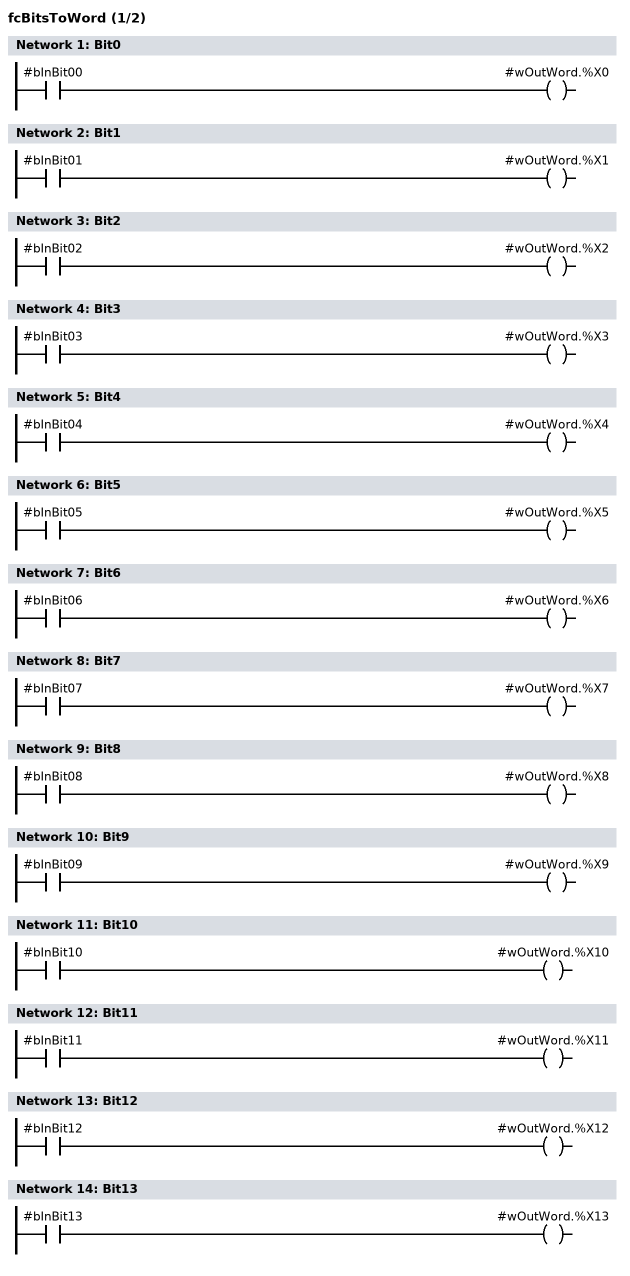
   RUNG wire#powerrail
      Contact( #bInBit00 )
      Coil( #wOutWord.%X0 )
   END_RUNG
   // the same network as SCL:
   #wOutWord.%X0 := #bInBit00;
END_REGION

REGION Network 2: Bit1
   RUNG wire#powerrail
      Contact( #bInBit01 )
      Coil( #wOutWord.%X1 )
   END_RUNG
   // the same network as SCL:
   #wOutWord.%X1 := #bInBit01;
END_REGION

REGION Network 3: Bit2
   RUNG wire#powerrail
      Contact( #bInBit02 )
      Coil( #wOutWord.%X2 )
   END_RUNG
   // the same network as SCL:
   #wOutWord.%X2 := #bInBit02;
END_REGION

REGION Network 4: Bit3
   RUNG wire#powerrail
      Contact( #bInBit03 )
      Coil( #wOutWord.%X3 )
   END_RUNG
   // the same network as SCL:
   #wOutWord.%X3 := #bInBit03;
END_REGION

REGION Network 5: Bit4
   RUNG wire#powerrail
      Contact( #bInBit04 )
      Coil( #wOutWord.%X4 )
   END_RUNG
   // the same network as SCL:
   #wOutWord.%X4 := #bInBit04;
END_REGION

REGION Network 6: Bit5
   RUNG wire#powerrail
      Contact( #bInBit05 )
      Coil( #wOutWord.%X5 )
   END_RUNG
   // the same network as SCL:
   #wOutWord.%X5 := #bInBit05;
END_REGION

REGION Network 7: Bit6
   RUNG wire#powerrail
      Contact( #bInBit06 )
      Coil( #wOutWord.%X6 )
   END_RUNG
   // the same network as SCL:
   #wOutWord.%X6 := #bInBit06;
END_REGION

REGION Network 8: Bit7
   RUNG wire#powerrail
      Contact( #bInBit07 )
      Coil( #wOutWord.%X7 )
   END_RUNG
   // the same network as SCL:
   #wOutWord.%X7 := #bInBit07;
END_REGION

REGION Network 9: Bit8
   RUNG wire#powerrail
      Contact( #bInBit08 )
      Coil( #wOutWord.%X8 )
   END_RUNG
   // the same network as SCL:
   #wOutWord.%X8 := #bInBit08;
END_REGION

REGION Network 10: Bit9
   RUNG wire#powerrail
      Contact( #bInBit09 )
      Coil( #wOutWord.%X9 )
   END_RUNG
   // the same network as SCL:
   #wOutWord.%X9 := #bInBit09;
END_REGION

REGION Network 11: Bit10
   RUNG wire#powerrail
      Contact( #bInBit10 )
      Coil( #wOutWord.%X10 )
   END_RUNG
   // the same network as SCL:
   #wOutWord.%X10 := #bInBit10;
END_REGION

REGION Network 12: Bit11
   RUNG wire#powerrail
      Contact( #bInBit11 )
      Coil( #wOutWord.%X11 )
   END_RUNG
   // the same network as SCL:
   #wOutWord.%X11 := #bInBit11;
END_REGION

REGION Network 13: Bit12
   RUNG wire#powerrail
      Contact( #bInBit12 )
      Coil( #wOutWord.%X12 )
   END_RUNG
   // the same network as SCL:
   #wOutWord.%X12 := #bInBit12;
END_REGION

REGION Network 14: Bit13
   RUNG wire#powerrail
      Contact( #bInBit13 )
      Coil( #wOutWord.%X13 )
   END_RUNG
   // the same network as SCL:
   #wOutWord.%X13 := #bInBit13;
END_REGION

REGION Network 15: Bit14
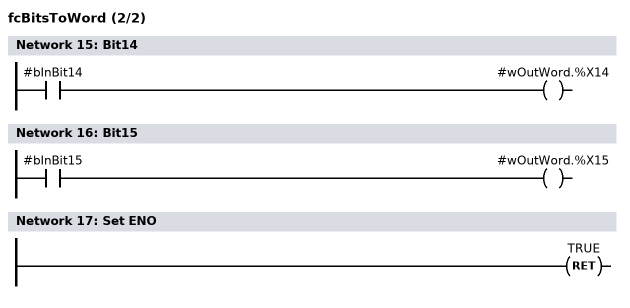
   RUNG wire#powerrail
      Contact( #bInBit14 )
      Coil( #wOutWord.%X14 )
   END_RUNG
   // the same network as SCL:
   #wOutWord.%X14 := #bInBit14;
END_REGION

REGION Network 16: Bit15
   RUNG wire#powerrail
      Contact( #bInBit15 )
      Coil( #wOutWord.%X15 )
   END_RUNG
   // the same network as SCL:
   #wOutWord.%X15 := #bInBit15;
END_REGION

REGION Network 17: Set ENO
   RUNG wire#powerrail
      ReturnCoil( TRUE )
   END_RUNG
   // the same network as SCL:
   ENO := TRUE;
   RETURN;
END_REGION
END_FUNCTION

FUNCTION "fcWordToBits" : Void   // FC303, LAD
TITLE = Breaks A Word Into Individual Bits
{ S7_Optimized_Access := 'TRUE' }
AUTHOR : DMC
FAMILY : LowLevel
VERSION : 0.1
   VAR_INPUT
      wInWord : Word;   // Word to be broken into individual bits
   END_VAR
   VAR_OUTPUT
      bOutBit00 : Bool;   // Bit 0
      bOutBit01 : Bool;   // Bit 1
      bOutBit02 : Bool;   // Bit 2
      bOutBit03 : Bool;   // Bit 3
      bOutBit04 : Bool;   // Bit 4
      bOutBit05 : Bool;   // Bit 5
      bOutBit06 : Bool;   // Bit 6
      bOutBit07 : Bool;   // Bit 7
      bOutBit08 : Bool;   // Bit 8
      bOutBit09 : Bool;   // Bit 9
      bOutBit10 : Bool;   // Bit 10
      bOutBit11 : Bool;   // Bit 11
      bOutBit12 : Bool;   // Bit 12
      bOutBit13 : Bool;   // Bit 13
      bOutBit14 : Bool;   // Bit 14
      bOutBit15 : Bool;   // Bit 15
   END_VAR
BEGIN

REGION Network 1: Bit0
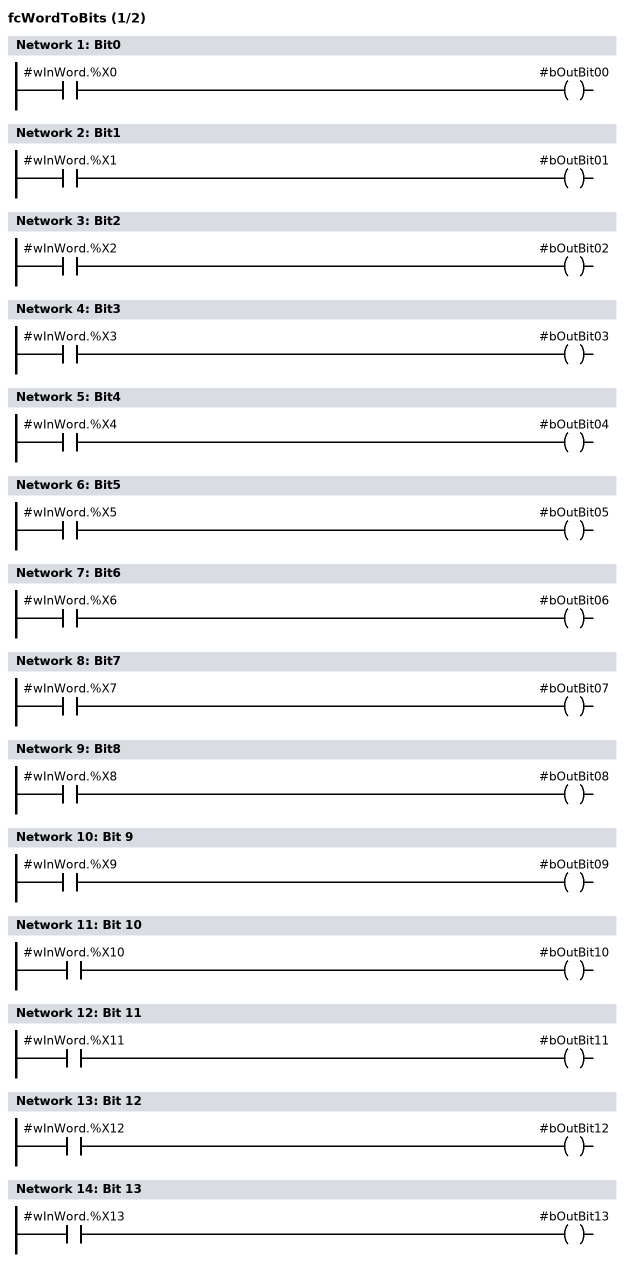
   RUNG wire#powerrail
      Contact( #wInWord.%X0 )
      Coil( #bOutBit00 )
   END_RUNG
   // the same network as SCL:
   #bOutBit00 := #wInWord.%X0;
END_REGION

REGION Network 2: Bit1
   RUNG wire#powerrail
      Contact( #wInWord.%X1 )
      Coil( #bOutBit01 )
   END_RUNG
   // the same network as SCL:
   #bOutBit01 := #wInWord.%X1;
END_REGION

REGION Network 3: Bit2
   RUNG wire#powerrail
      Contact( #wInWord.%X2 )
      Coil( #bOutBit02 )
   END_RUNG
   // the same network as SCL:
   #bOutBit02 := #wInWord.%X2;
END_REGION

REGION Network 4: Bit3
   RUNG wire#powerrail
      Contact( #wInWord.%X3 )
      Coil( #bOutBit03 )
   END_RUNG
   // the same network as SCL:
   #bOutBit03 := #wInWord.%X3;
END_REGION

REGION Network 5: Bit4
   RUNG wire#powerrail
      Contact( #wInWord.%X4 )
      Coil( #bOutBit04 )
   END_RUNG
   // the same network as SCL:
   #bOutBit04 := #wInWord.%X4;
END_REGION

REGION Network 6: Bit5
   RUNG wire#powerrail
      Contact( #wInWord.%X5 )
      Coil( #bOutBit05 )
   END_RUNG
   // the same network as SCL:
   #bOutBit05 := #wInWord.%X5;
END_REGION

REGION Network 7: Bit6
   RUNG wire#powerrail
      Contact( #wInWord.%X6 )
      Coil( #bOutBit06 )
   END_RUNG
   // the same network as SCL:
   #bOutBit06 := #wInWord.%X6;
END_REGION

REGION Network 8: Bit7
   RUNG wire#powerrail
      Contact( #wInWord.%X7 )
      Coil( #bOutBit07 )
   END_RUNG
   // the same network as SCL:
   #bOutBit07 := #wInWord.%X7;
END_REGION

REGION Network 9: Bit8
   RUNG wire#powerrail
      Contact( #wInWord.%X8 )
      Coil( #bOutBit08 )
   END_RUNG
   // the same network as SCL:
   #bOutBit08 := #wInWord.%X8;
END_REGION

REGION Network 10: Bit 9
   RUNG wire#powerrail
      Contact( #wInWord.%X9 )
      Coil( #bOutBit09 )
   END_RUNG
   // the same network as SCL:
   #bOutBit09 := #wInWord.%X9;
END_REGION

REGION Network 11: Bit 10
   RUNG wire#powerrail
      Contact( #wInWord.%X10 )
      Coil( #bOutBit10 )
   END_RUNG
   // the same network as SCL:
   #bOutBit10 := #wInWord.%X10;
END_REGION

REGION Network 12: Bit 11
   RUNG wire#powerrail
      Contact( #wInWord.%X11 )
      Coil( #bOutBit11 )
   END_RUNG
   // the same network as SCL:
   #bOutBit11 := #wInWord.%X11;
END_REGION

REGION Network 13: Bit 12
   RUNG wire#powerrail
      Contact( #wInWord.%X12 )
      Coil( #bOutBit12 )
   END_RUNG
   // the same network as SCL:
   #bOutBit12 := #wInWord.%X12;
END_REGION

REGION Network 14: Bit 13
   RUNG wire#powerrail
      Contact( #wInWord.%X13 )
      Coil( #bOutBit13 )
   END_RUNG
   // the same network as SCL:
   #bOutBit13 := #wInWord.%X13;
END_REGION

REGION Network 15: Bit 14
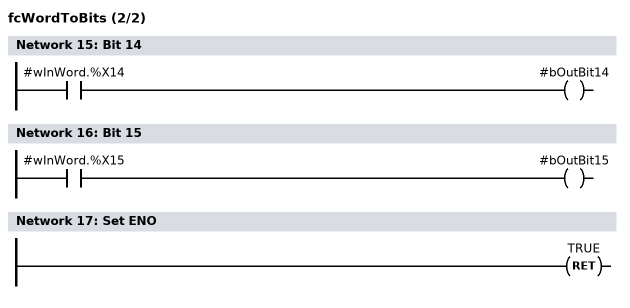
   RUNG wire#powerrail
      Contact( #wInWord.%X14 )
      Coil( #bOutBit14 )
   END_RUNG
   // the same network as SCL:
   #bOutBit14 := #wInWord.%X14;
END_REGION

REGION Network 16: Bit 15
   RUNG wire#powerrail
      Contact( #wInWord.%X15 )
      Coil( #bOutBit15 )
   END_RUNG
   // the same network as SCL:
   #bOutBit15 := #wInWord.%X15;
END_REGION

REGION Network 17: Set ENO
   RUNG wire#powerrail
      ReturnCoil( TRUE )
   END_RUNG
   // the same network as SCL:
   ENO := TRUE;
   RETURN;
END_REGION
END_FUNCTION

// folder: Resources/fbVFD/Resources/HMI

FUNCTION_BLOCK "fbErrorScroller"   // FB330, LAD
TITLE = Scrolls through the error codes for display on the HMI
{ S7_Optimized_Access := 'TRUE' }
AUTHOR : DMC
FAMILY : Error
VERSION : 0.1
   VAR_INPUT
      bInError01 : Bool;   // Error 1 In Error Array
      bInError02 : Bool;   // Error 2 In Error Array
      bInError03 : Bool;   // Error 3 In Error Array
      bInError04 : Bool;   // Error 4 In Error Array
      bInError05 : Bool;   // Error 5 In Error Array
      bInError06 : Bool;   // Error 6 In Error Array
      bInError07 : Bool;   // Error 7 In Error Array
      bInError08 : Bool;   // Error 8 In Error Array
      bInError09 : Bool;   // Error 9 In Error Array
      bInError10 : Bool;   // Error 10 In Error Array
      bInError11 : Bool;   // Error 11 In Error Array
      bInError12 : Bool;   // Error 12 In Error Array
      bInError13 : Bool;   // Error 13 In Error Array
      bInError14 : Bool;   // Error 14 In Error Array
      bInError15 : Bool;   // Error 15 In Error Array
      bInError16 : Bool;   // Error 16 In Error Array
      bInError17 : Bool;   // Error 17 In Error Array
      bInError18 : Bool;   // Error 18 In Error Array
      bInError19 : Bool;   // Error 19 In Error Array
      bInError20 : Bool;   // Error 20 In Error Array
      bInError21 : Bool;   // Error 21 In Error Array
      bInError22 : Bool;   // Error 22 In Error Array
      bInError23 : Bool;   // Error 23 In Error Array
      bInError24 : Bool;   // Error 24 In Error Array
      bInError25 : Bool;   // Error 25 In Error Array
      bInError26 : Bool;   // Error 26 In Error Array
      bInError27 : Bool;   // Error 27 In Error Array
      bInError28 : Bool;   // Error 28 In Error Array
      bInError29 : Bool;   // Error 29 In Error Array
      bInError30 : Bool;   // Error 30 In Error Array
   END_VAR
   VAR_OUTPUT
      bOutErrorExists : Bool;   // An Error Exists
      iOutScrollingErrorNumber : Int;   // Current Index when scrolling through errors
   END_VAR
   VAR
      TON_ErrorDelay : TON_TIME;   // Delay between each scroll for a new error
      abErrors : Array[#ciIndexLow..#ciIndexHigh] of Bool;
      iNextScrollNum : Int := 1;   // Index of next error position
      iErrorsScrollNum : Int := 1;   // Index of current error position
      bScrolling : Bool;   // Indicates we are scrolling
      bTON_ErrorDelay : Bool;
   END_VAR
   VAR_TEMP
      bErrorExists : Bool;   // Error Exists
   END_VAR
   VAR CONSTANT
      ciNoErrrors : Int := 0;
      ciIndexLow : Int := 1;
      ciIndexHigh : Int := 30;
   END_VAR
   VAR_TEMP   // added for the SCL form of the ladder/FBD networks
      _w1 : Bool;
   END_VAR
BEGIN

REGION Network 1: Check for valid array indexes
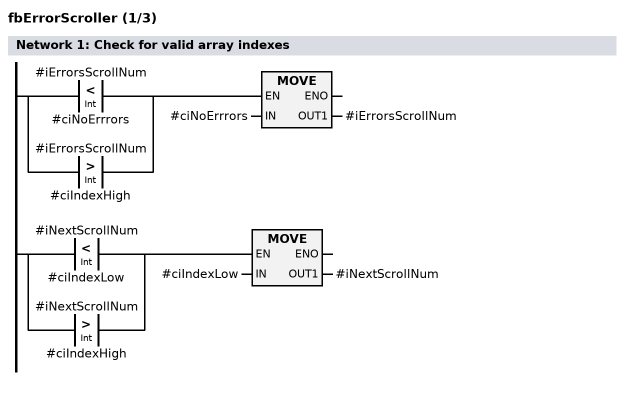
   RUNG wire#powerrail
      { S7_Templates := "SrcType := Int" } LT_Contact(in1 := #iErrorsScrollNum, in2 := #ciNoErrrors)
      wire#w1
      Move(in := #ciNoErrrors, out1 => #iErrorsScrollNum)
   END_RUNG
   RUNG wire#powerrail
      { S7_Templates := "SrcType := Int" } GT_Contact(in1 := #iErrorsScrollNum, in2 := #ciIndexHigh)
   END_RUNG wire#w1
   RUNG wire#powerrail
      { S7_Templates := "SrcType := Int" } LT_Contact(in1 := #iNextScrollNum, in2 := #ciIndexLow)
      wire#w2
      Move(in := #ciIndexLow, out1 => #iNextScrollNum)
   END_RUNG
   RUNG wire#powerrail
      { S7_Templates := "SrcType := Int" } GT_Contact(in1 := #iNextScrollNum, in2 := #ciIndexHigh)
   END_RUNG wire#w2
   // the same network as SCL:
   IF (#iErrorsScrollNum < #ciNoErrrors) OR (#iErrorsScrollNum > #ciIndexHigh) THEN
       #iErrorsScrollNum := #ciNoErrrors;
   END_IF;
   IF (#iNextScrollNum < #ciIndexLow) OR (#iNextScrollNum > #ciIndexHigh) THEN
       #iNextScrollNum := #ciIndexLow;
   END_IF;
END_REGION

REGION Network 2: Check if error exists
   // OR all of the possible errors. If any error Exists, SET bErrorExists
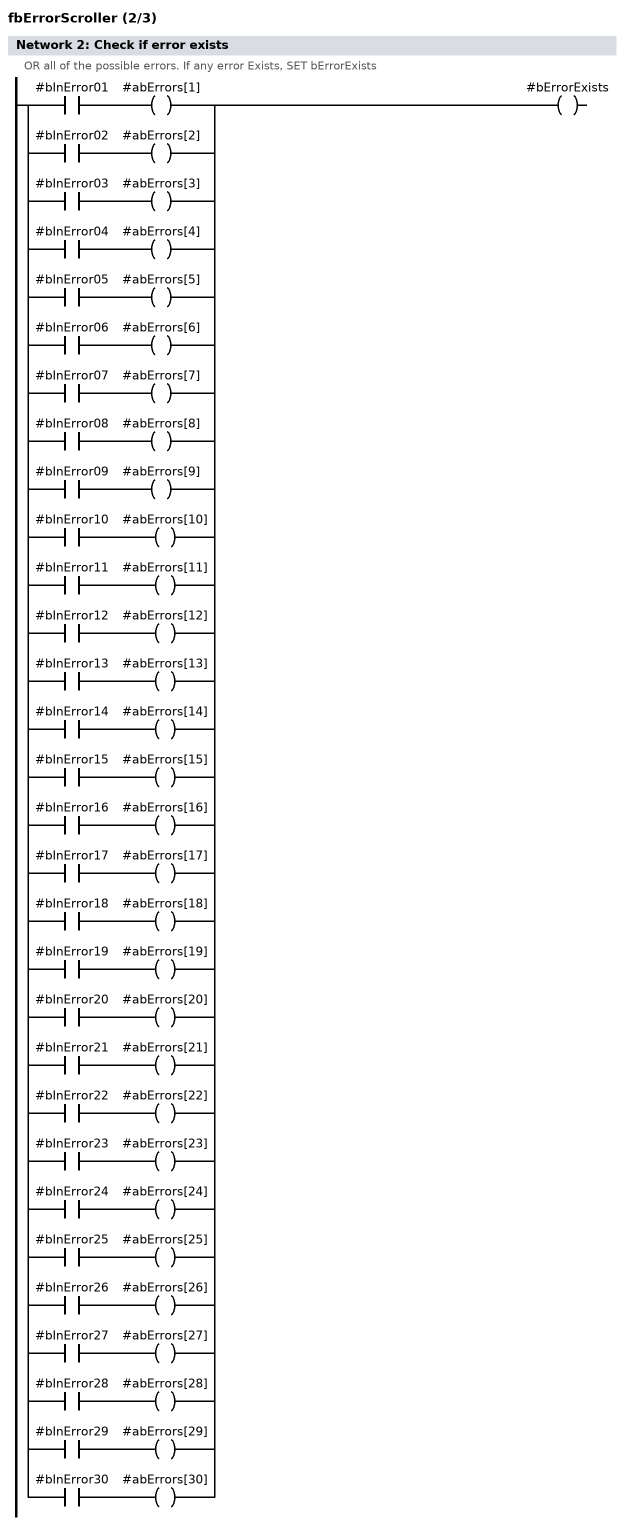
   RUNG wire#powerrail
      Contact( #bInError01 )
      Coil( #abErrors[1] )
      wire#w1
      Coil( #bErrorExists )
   END_RUNG
   RUNG wire#powerrail
      Contact( #bInError02 )
      Coil( #abErrors[2] )
   END_RUNG wire#w1
   RUNG wire#powerrail
      Contact( #bInError03 )
      Coil( #abErrors[3] )
   END_RUNG wire#w1
   RUNG wire#powerrail
      Contact( #bInError04 )
      Coil( #abErrors[4] )
   END_RUNG wire#w1
   RUNG wire#powerrail
      Contact( #bInError05 )
      Coil( #abErrors[5] )
   END_RUNG wire#w1
   RUNG wire#powerrail
      Contact( #bInError06 )
      Coil( #abErrors[6] )
   END_RUNG wire#w1
   RUNG wire#powerrail
      Contact( #bInError07 )
      Coil( #abErrors[7] )
   END_RUNG wire#w1
   RUNG wire#powerrail
      Contact( #bInError08 )
      Coil( #abErrors[8] )
   END_RUNG wire#w1
   RUNG wire#powerrail
      Contact( #bInError09 )
      Coil( #abErrors[9] )
   END_RUNG wire#w1
   RUNG wire#powerrail
      Contact( #bInError10 )
      Coil( #abErrors[10] )
   END_RUNG wire#w1
   RUNG wire#powerrail
      Contact( #bInError11 )
      Coil( #abErrors[11] )
   END_RUNG wire#w1
   RUNG wire#powerrail
      Contact( #bInError12 )
      Coil( #abErrors[12] )
   END_RUNG wire#w1
   RUNG wire#powerrail
      Contact( #bInError13 )
      Coil( #abErrors[13] )
   END_RUNG wire#w1
   RUNG wire#powerrail
      Contact( #bInError14 )
      Coil( #abErrors[14] )
   END_RUNG wire#w1
   RUNG wire#powerrail
      Contact( #bInError15 )
      Coil( #abErrors[15] )
   END_RUNG wire#w1
   RUNG wire#powerrail
      Contact( #bInError16 )
      Coil( #abErrors[16] )
   END_RUNG wire#w1
   RUNG wire#powerrail
      Contact( #bInError17 )
      Coil( #abErrors[17] )
   END_RUNG wire#w1
   RUNG wire#powerrail
      Contact( #bInError18 )
      Coil( #abErrors[18] )
   END_RUNG wire#w1
   RUNG wire#powerrail
      Contact( #bInError19 )
      Coil( #abErrors[19] )
   END_RUNG wire#w1
   RUNG wire#powerrail
      Contact( #bInError20 )
      Coil( #abErrors[20] )
   END_RUNG wire#w1
   RUNG wire#powerrail
      Contact( #bInError21 )
      Coil( #abErrors[21] )
   END_RUNG wire#w1
   RUNG wire#powerrail
      Contact( #bInError22 )
      Coil( #abErrors[22] )
   END_RUNG wire#w1
   RUNG wire#powerrail
      Contact( #bInError23 )
      Coil( #abErrors[23] )
   END_RUNG wire#w1
   RUNG wire#powerrail
      Contact( #bInError24 )
      Coil( #abErrors[24] )
   END_RUNG wire#w1
   RUNG wire#powerrail
      Contact( #bInError25 )
      Coil( #abErrors[25] )
   END_RUNG wire#w1
   RUNG wire#powerrail
      Contact( #bInError26 )
      Coil( #abErrors[26] )
   END_RUNG wire#w1
   RUNG wire#powerrail
      Contact( #bInError27 )
      Coil( #abErrors[27] )
   END_RUNG wire#w1
   RUNG wire#powerrail
      Contact( #bInError28 )
      Coil( #abErrors[28] )
   END_RUNG wire#w1
   RUNG wire#powerrail
      Contact( #bInError29 )
      Coil( #abErrors[29] )
   END_RUNG wire#w1
   RUNG wire#powerrail
      Contact( #bInError30 )
      Coil( #abErrors[30] )
   END_RUNG wire#w1
   // the same network as SCL:
   #abErrors[1] := #bInError01;
   #abErrors[2] := #bInError02;
   #abErrors[3] := #bInError03;
   #abErrors[4] := #bInError04;
   #abErrors[5] := #bInError05;
   #abErrors[6] := #bInError06;
   #abErrors[7] := #bInError07;
   #abErrors[8] := #bInError08;
   #abErrors[9] := #bInError09;
   #abErrors[10] := #bInError10;
   #abErrors[11] := #bInError11;
   #abErrors[12] := #bInError12;
   #abErrors[13] := #bInError13;
   #abErrors[14] := #bInError14;
   #abErrors[15] := #bInError15;
   #abErrors[16] := #bInError16;
   #abErrors[17] := #bInError17;
   #abErrors[18] := #bInError18;
   #abErrors[19] := #bInError19;
   #abErrors[20] := #bInError20;
   #abErrors[21] := #bInError21;
   #abErrors[22] := #bInError22;
   #abErrors[23] := #bInError23;
   #abErrors[24] := #bInError24;
   #abErrors[25] := #bInError25;
   #abErrors[26] := #bInError26;
   #abErrors[27] := #bInError27;
   #abErrors[28] := #bInError28;
   #abErrors[29] := #bInError29;
   #abErrors[30] := #bInError30;
   #bErrorExists := #bInError01 OR #bInError02 OR #bInError03 OR #bInError04 OR #bInError05 OR #bInError06 OR #bInError07 OR #bInError08 OR #bInError09 OR #bInError10 OR #bInError11 OR #bInError12 OR #bInError13 OR #bInError14 OR #bInError15 OR #bInError16 OR #bInError17 OR #bInError18 OR #bInError19 OR #bInError20 OR #bInError21 OR #bInError22 OR #bInError23 OR #bInError24 OR #bInError25 OR #bInError26 OR #bInError27 OR #bInError28 OR #bInError29 OR #bInError30;
END_REGION

REGION Network 3: Timer to change displayed error
   // ============================ Scroll errors on HMI ========================
   // Timed delay
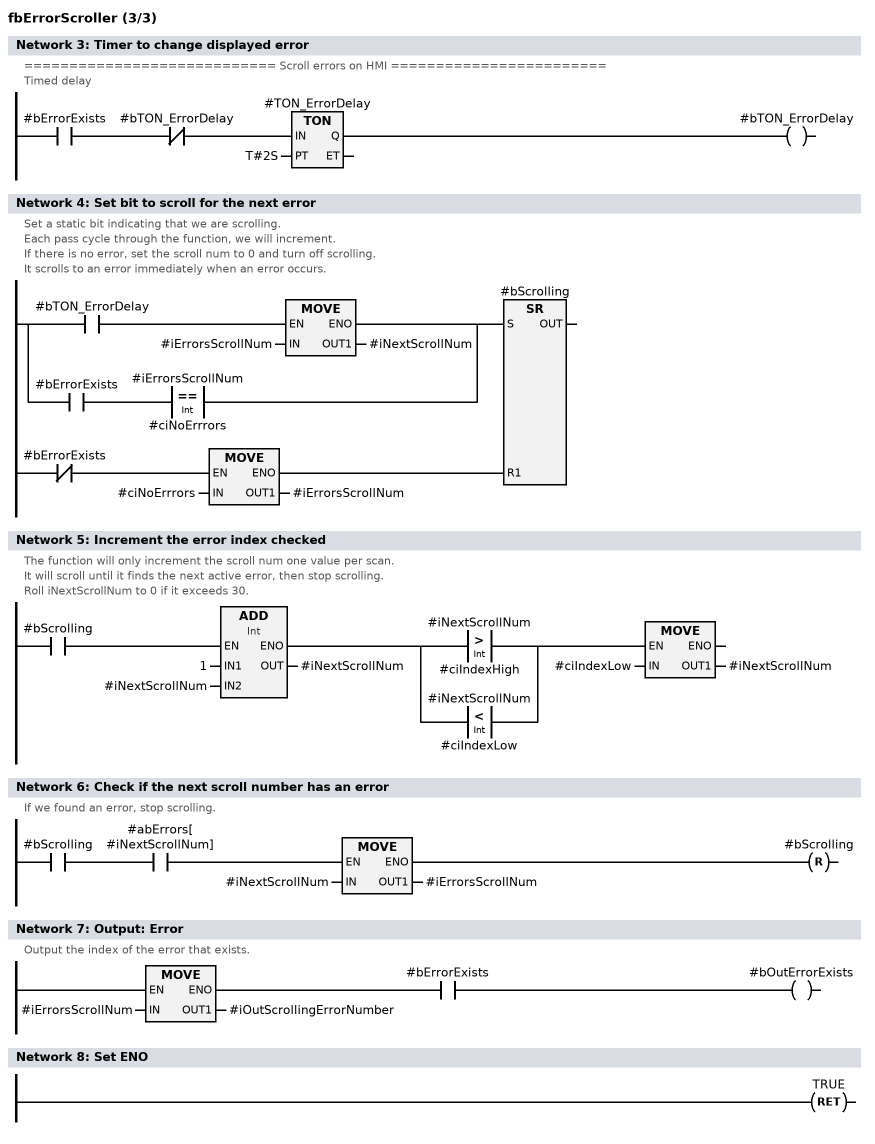
   #TON_ErrorDelay(IN := #bErrorExists AND NOT #bTON_ErrorDelay, PT := T#2S);   // TON
   #bTON_ErrorDelay := #TON_ErrorDelay.Q;
END_REGION

REGION Network 4: Set bit to scroll for the next error
   // Set a static bit indicating that we are scrolling.  
   // Each pass cycle through the function, we will increment.  
   // If there is no error, set the scroll num to 0 and turn off scrolling.  
   // It scrolls to an error immediately when an error occurs.
   RUNG wire#powerrail
      Contact( #bTON_ErrorDelay )
      { S7_GenerateENO := "TRUE" } Move(in := #iErrorsScrollNum, out1 => #iNextScrollNum)
      wire#w1
      S_SR(operand := #bScrolling, r1 := wire#w2)
   END_RUNG
   RUNG wire#powerrail
      Contact( #bErrorExists )
      { S7_Templates := "SrcType := Int" } EQ_Contact(in1 := #iErrorsScrollNum, in2 := #ciNoErrrors)
   END_RUNG wire#w1
   RUNG wire#powerrail
      I_Contact( #bErrorExists )
      { S7_GenerateENO := "TRUE" } Move(in := #ciNoErrrors, out1 => #iErrorsScrollNum)
   END_RUNG wire#w2
   // the same network as SCL:
   // ENO of a box is taken as its EN; it also drops when the box reports an error
   IF #bTON_ErrorDelay THEN #iNextScrollNum := #iErrorsScrollNum; END_IF;
   #_w1 := #bTON_ErrorDelay OR (#bErrorExists AND (#iErrorsScrollNum = #ciNoErrrors));
   IF NOT #bErrorExists THEN #iErrorsScrollNum := #ciNoErrrors; END_IF;
   IF #_w1 THEN
       #bScrolling := TRUE;   // SR flip-flop
   END_IF;
   IF NOT #bErrorExists THEN #bScrolling := FALSE; END_IF;
END_REGION

REGION Network 5: Increment the error index checked
   // The function will only increment the scroll num one value per scan.  
   // It will scroll until it finds the next active error, then stop scrolling.  
   // Roll iNextScrollNum to 0 if it exceeds 30.
   RUNG wire#powerrail
      Contact( #bScrolling )
      { S7_Templates := "SrcType := Int"; S7_GenerateENO := "TRUE" } Add(in1 := 1, in2 := #iNextScrollNum, out => #iNextScrollNum)
      wire#w1
      { S7_Templates := "SrcType := Int" } GT_Contact(in1 := #iNextScrollNum, in2 := #ciIndexHigh)
      wire#w2
      { S7_GenerateENO := "TRUE" } Move(in := #ciIndexLow, out1 => #iNextScrollNum)
   END_RUNG
   RUNG wire#w1
      { S7_Templates := "SrcType := Int" } LT_Contact(in1 := #iNextScrollNum, in2 := #ciIndexLow)
   END_RUNG wire#w2
   // the same network as SCL:
   // ENO of a box is taken as its EN; it also drops when the box reports an error
   IF #bScrolling THEN #iNextScrollNum := 1 + #iNextScrollNum; END_IF;
   IF #bScrolling AND ((#iNextScrollNum > #ciIndexHigh) OR (#iNextScrollNum < #ciIndexLow)) THEN
       #iNextScrollNum := #ciIndexLow;
   END_IF;
END_REGION

REGION Network 6: Check if the next scroll number has an error
   // If we found an error, stop scrolling.
   RUNG wire#powerrail
      Contact( #bScrolling )
      Contact( #abErrors[#iNextScrollNum] )
      { S7_GenerateENO := "TRUE" } Move(in := #iNextScrollNum, out1 => #iErrorsScrollNum)
      R_Coil( #bScrolling )
   END_RUNG
   // the same network as SCL:
   // ENO of a box is taken as its EN; it also drops when the box reports an error
   IF #bScrolling AND #abErrors[#iNextScrollNum] THEN
       #iErrorsScrollNum := #iNextScrollNum;
       #bScrolling := FALSE;
   END_IF;
END_REGION

REGION Network 7: Output: Error
   // Output the index of the error that exists.
   RUNG wire#powerrail
      { S7_GenerateENO := "TRUE" } Move(in := #iErrorsScrollNum, out1 => #iOutScrollingErrorNumber)
      Contact( #bErrorExists )
      Coil( #bOutErrorExists )
   END_RUNG
   // the same network as SCL:
   // ENO of a box is taken as its EN; it also drops when the box reports an error
   #iOutScrollingErrorNumber := #iErrorsScrollNum;
   #bOutErrorExists := #bErrorExists;
END_REGION

REGION Network 8: Set ENO
   RUNG wire#powerrail
      ReturnCoil( TRUE )
   END_RUNG
   // the same network as SCL:
   ENO := TRUE;
   RETURN;
END_REGION
END_FUNCTION_BLOCK

FUNCTION "fcHMIBitEnable" : Void   // FC329, LAD
TITLE = Handles an async reading of an HMI bit to avoid race conditions, includes an enable bit
{ S7_Optimized_Access := 'TRUE' }
VERSION : 0.1
   VAR_INPUT
      bInToggle : Bool;
      bInLatch : Bool;
      bInEnable : Bool;
   END_VAR
   VAR_OUTPUT
      bOutEnable : Bool;
   END_VAR
   VAR_IN_OUT
      bInOutHMI : Bool;
      bInOutPLC : Bool;
   END_VAR
   VAR_TEMP   // added for the SCL form of the ladder/FBD networks
      _w1 : Bool;
   END_VAR
BEGIN

REGION Network 1: If not latching or toggling, reset the PLC bit every scan
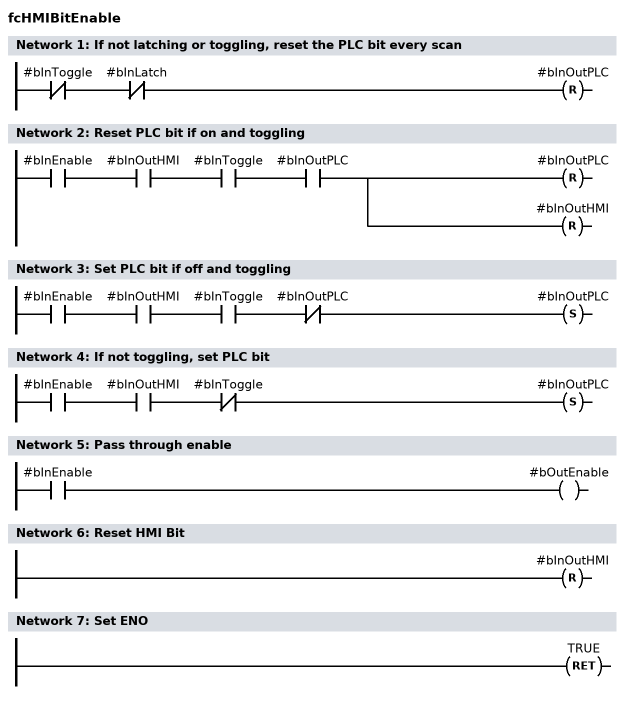
   RUNG wire#powerrail
      I_Contact( #bInToggle )
      I_Contact( #bInLatch )
      R_Coil( #bInOutPLC )
   END_RUNG
   // the same network as SCL:
   IF NOT #bInToggle AND NOT #bInLatch THEN #bInOutPLC := FALSE; END_IF;
END_REGION

REGION Network 2: Reset PLC bit if on and toggling
   RUNG wire#powerrail
      Contact( #bInEnable )
      Contact( #bInOutHMI )
      Contact( #bInToggle )
      Contact( #bInOutPLC )
      wire#w1
      R_Coil( #bInOutPLC )
   END_RUNG
   RUNG wire#w1
      R_Coil( #bInOutHMI )
   END_RUNG
   // the same network as SCL:
   #_w1 := #bInEnable AND #bInOutHMI AND #bInToggle AND #bInOutPLC;
   IF #_w1 THEN
       #bInOutPLC := FALSE;
       #bInOutHMI := FALSE;
   END_IF;
END_REGION

REGION Network 3: Set PLC bit if off and toggling
   RUNG wire#powerrail
      Contact( #bInEnable )
      Contact( #bInOutHMI )
      Contact( #bInToggle )
      I_Contact( #bInOutPLC )
      S_Coil( #bInOutPLC )
   END_RUNG
   // the same network as SCL:
   IF #bInEnable AND #bInOutHMI AND #bInToggle AND NOT #bInOutPLC THEN #bInOutPLC := TRUE; END_IF;
END_REGION

REGION Network 4: If not toggling, set PLC bit
   RUNG wire#powerrail
      Contact( #bInEnable )
      Contact( #bInOutHMI )
      I_Contact( #bInToggle )
      S_Coil( #bInOutPLC )
   END_RUNG
   // the same network as SCL:
   IF #bInEnable AND #bInOutHMI AND NOT #bInToggle THEN #bInOutPLC := TRUE; END_IF;
END_REGION

REGION Network 5: Pass through enable
   RUNG wire#powerrail
      Contact( #bInEnable )
      Coil( #bOutEnable )
   END_RUNG
   // the same network as SCL:
   #bOutEnable := #bInEnable;
END_REGION

REGION Network 6: Reset HMI Bit
   RUNG wire#powerrail
      R_Coil( #bInOutHMI )
   END_RUNG
   // the same network as SCL:
   #bInOutHMI := FALSE;
END_REGION

REGION Network 7: Set ENO
   RUNG wire#powerrail
      ReturnCoil( TRUE )
   END_RUNG
   // the same network as SCL:
   ENO := TRUE;
   RETURN;
END_REGION
END_FUNCTION

FUNCTION "fcSetHMIStatusSimulation" : Void   // FC333, LAD
TITLE = Sets HMI Status
{ S7_Optimized_Access := 'TRUE' }
VERSION : 0.1
// Wrapper function for setting the HMI status of a device
// 
// In order of priority:
// 1. E-stop
// 2. Error
// 3. Forward/Work Position
// 4. Reverse/Home Position
// 5. Forward/Work On
// 6. Reverse/Home On
// 7. None
   VAR_INPUT
      bInEstop : Bool;
      bInError : Bool;
      bInForwardWork : Bool;
      bInReverseHome : Bool;
      bInOnForwardWork : Bool;
      bInOnReverseHome : Bool;
      bInSimulate : Bool;
   END_VAR
   VAR_OUTPUT
      iOutStatus : Int;
   END_VAR
BEGIN

REGION Network 1: Set Reverse/Home On
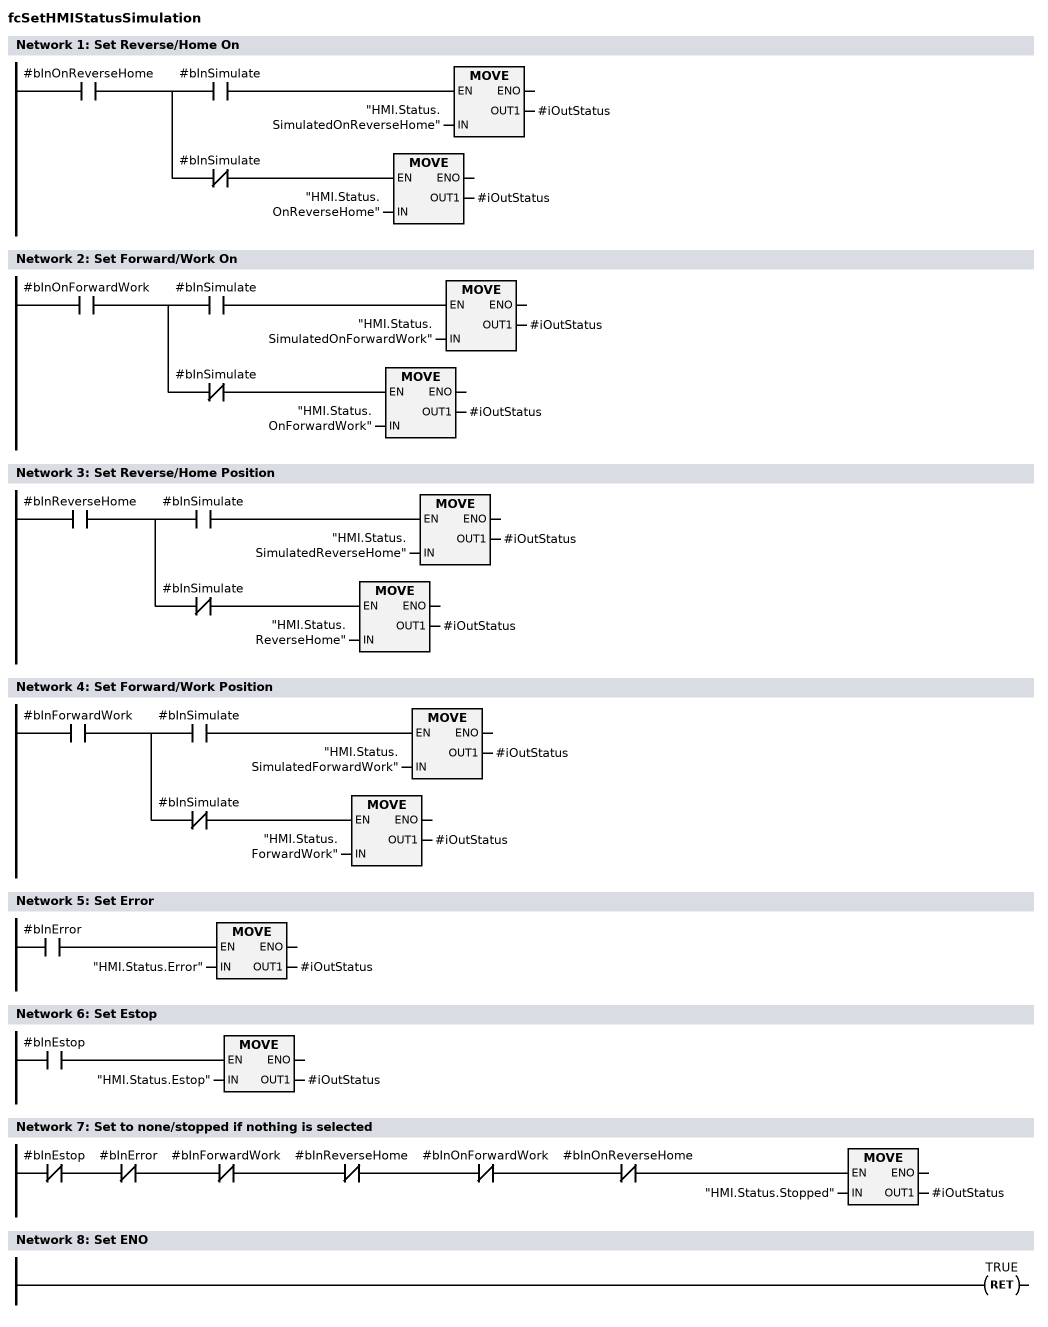
   RUNG wire#powerrail
      Contact( #bInOnReverseHome )
      wire#w1
      Contact( #bInSimulate )
      Move(in := "HMI.Status.SimulatedOnReverseHome", out1 => #iOutStatus)
   END_RUNG
   RUNG wire#w1
      I_Contact( #bInSimulate )
      Move(in := "HMI.Status.OnReverseHome", out1 => #iOutStatus)
   END_RUNG
   // the same network as SCL:
   IF #bInOnReverseHome AND #bInSimulate THEN #iOutStatus := "HMI.Status.SimulatedOnReverseHome"; END_IF;
   IF #bInOnReverseHome AND NOT #bInSimulate THEN #iOutStatus := "HMI.Status.OnReverseHome"; END_IF;
END_REGION

REGION Network 2: Set Forward/Work On
   RUNG wire#powerrail
      Contact( #bInOnForwardWork )
      wire#w1
      Contact( #bInSimulate )
      Move(in := "HMI.Status.SimulatedOnForwardWork", out1 => #iOutStatus)
   END_RUNG
   RUNG wire#w1
      I_Contact( #bInSimulate )
      Move(in := "HMI.Status.OnForwardWork", out1 => #iOutStatus)
   END_RUNG
   // the same network as SCL:
   IF #bInOnForwardWork AND #bInSimulate THEN #iOutStatus := "HMI.Status.SimulatedOnForwardWork"; END_IF;
   IF #bInOnForwardWork AND NOT #bInSimulate THEN #iOutStatus := "HMI.Status.OnForwardWork"; END_IF;
END_REGION

REGION Network 3: Set Reverse/Home Position
   RUNG wire#powerrail
      Contact( #bInReverseHome )
      wire#w1
      Contact( #bInSimulate )
      Move(in := "HMI.Status.SimulatedReverseHome", out1 => #iOutStatus)
   END_RUNG
   RUNG wire#w1
      I_Contact( #bInSimulate )
      Move(in := "HMI.Status.ReverseHome", out1 => #iOutStatus)
   END_RUNG
   // the same network as SCL:
   IF #bInReverseHome AND #bInSimulate THEN #iOutStatus := "HMI.Status.SimulatedReverseHome"; END_IF;
   IF #bInReverseHome AND NOT #bInSimulate THEN #iOutStatus := "HMI.Status.ReverseHome"; END_IF;
END_REGION

REGION Network 4: Set Forward/Work Position
   RUNG wire#powerrail
      Contact( #bInForwardWork )
      wire#w1
      Contact( #bInSimulate )
      Move(in := "HMI.Status.SimulatedForwardWork", out1 => #iOutStatus)
   END_RUNG
   RUNG wire#w1
      I_Contact( #bInSimulate )
      Move(in := "HMI.Status.ForwardWork", out1 => #iOutStatus)
   END_RUNG
   // the same network as SCL:
   IF #bInForwardWork AND #bInSimulate THEN #iOutStatus := "HMI.Status.SimulatedForwardWork"; END_IF;
   IF #bInForwardWork AND NOT #bInSimulate THEN #iOutStatus := "HMI.Status.ForwardWork"; END_IF;
END_REGION

REGION Network 5: Set Error
   RUNG wire#powerrail
      Contact( #bInError )
      Move(in := "HMI.Status.Error", out1 => #iOutStatus)
   END_RUNG
   // the same network as SCL:
   IF #bInError THEN #iOutStatus := "HMI.Status.Error"; END_IF;
END_REGION

REGION Network 6: Set Estop
   RUNG wire#powerrail
      Contact( #bInEstop )
      Move(in := "HMI.Status.Estop", out1 => #iOutStatus)
   END_RUNG
   // the same network as SCL:
   IF #bInEstop THEN #iOutStatus := "HMI.Status.Estop"; END_IF;
END_REGION

REGION Network 7: Set to none/stopped if nothing is selected
   RUNG wire#powerrail
      I_Contact( #bInEstop )
      I_Contact( #bInError )
      I_Contact( #bInForwardWork )
      I_Contact( #bInReverseHome )
      I_Contact( #bInOnForwardWork )
      I_Contact( #bInOnReverseHome )
      Move(in := "HMI.Status.Stopped", out1 => #iOutStatus)
   END_RUNG
   // the same network as SCL:
   IF NOT #bInEstop AND NOT #bInError AND NOT #bInForwardWork AND NOT #bInReverseHome AND NOT #bInOnForwardWork AND NOT #bInOnReverseHome THEN
       #iOutStatus := "HMI.Status.Stopped";
   END_IF;
END_REGION

REGION Network 8: Set ENO
   RUNG wire#powerrail
      ReturnCoil( TRUE )
   END_RUNG
   // the same network as SCL:
   ENO := TRUE;
   RETURN;
END_REGION
END_FUNCTION

// ===== library types =====

TYPE "udtDriveTestParams"
   STRUCT
      bEStop : Bool;   // 1 = Emergency stop the drive
      rTargetSpeed : Real;   // Target speed for drive
      bCommandForward : Bool;   // Commands the drive to run forward
      bCommandReverse : Bool;   // Commands the drive to run in reverse
      bResetError : Bool;   // Clear any errors on the drive
      rActualSpeed : Real;   // Actual speed reported from drive
      bActiveError : Bool;   // Drive Error Active
   END_STRUCT;
END_TYPE

// folder: Data Types/Error

TYPE "udtError_SolenoidValve"
VERSION : 0.1
   STRUCT
      NoHomeFeedback : Bool;   // Home position feedback not active
      NoWorkFeedback : Bool;   // Work position feedback not active
      HomeFeedbackStillActive : Bool;   // Home position feedback still active
      WorkFeedbackStillActive : Bool;   // Work position feedback still active
   END_STRUCT;
END_TYPE

TYPE "udtError_AnalogInput"
VERSION : 0.1
   STRUCT
      LowLowAlarm : Bool;   // Value below low low set point
      HighHighAlarm : Bool;   // Value above high high set point
      Invalid : Bool;   // Invalid input valid
   END_STRUCT;
END_TYPE

// folder: Data Types/HMI

TYPE "udtHMI_PushButton"
VERSION : 0.1
   STRUCT
      bPB : Bool;   // Push Button
      bPBEN : Bool;   // Push Button Control Enable
      iPBLT : Int;   // used to determine button color
      sTitle : String;   // Button title
   END_STRUCT;
END_TYPE

// folder: Library Data Types/Devices/HMI

TYPE "udtHMI_DigitalOutput"
VERSION : 0.1
   STRUCT
      iMode : Int;   // Current mode
      bCommand : Bool;   // Output command value
      bCommandAuto : Bool;   // Auto mode command value
      bInterlock : Bool;   // Analog output is interlocked
      On : "udtHMI_PushButton";   // PB: Turn output on in manual mode
      Off : "udtHMI_PushButton";   // PB: Turn output off in manual mode
   END_STRUCT;
END_TYPE

TYPE "udtHMI_SolenoidValve"
VERSION : 0.1
   STRUCT
      iMode : Int;   // Current mode
      iErrorCode : Int;   // Error code
      iStatus : Int;   // Status for HMI display
      ResetError : "udtHMI_PushButton";   // PB: Reset block errors
      Home : "udtHMI_PushButton";   // PB: Move to home in manual mode
      Work : "udtHMI_PushButton";   // PB: Move to work in manual mode
      bHomeOn : Bool;   // Home command is on
      bWorkOn : Bool;   // Work command is on
      bSignalHome : Bool;   // Home feedback
      bSignalWork : Bool;   // Work feedback
      bError : Bool;   // Error status
      bInterlock : Bool;   // Valve interlocked
   END_STRUCT;
END_TYPE

TYPE "udtHMI_AnalogInput"
VERSION : 0.1
   STRUCT
      iMode : Int;   // Current mode
      iErrorCode : Int;   // Error code
      iStatus : Int;   // Overall HMI Status
      rActiveValue : Real;   // Used Value, Input or Override
      rInputValue : Real;   // Input Value
      rManualValue : Real;   // Manual mode simulated value
      ResetError : "udtHMI_PushButton";   // PB: Reset block errors
      bError : Bool;   // Overall error
   END_STRUCT;
END_TYPE

TYPE "udtHMI_DigitalInput"
VERSION : 0.1
   STRUCT
      iMode : Int;   // Current mode
      bOn : Bool;   // Status of the sensor
      bOnActual : Bool;   // Status of the physical sensor
      On : "udtHMI_PushButton";   // PB: Turn input on in manual mode
      Off : "udtHMI_PushButton";   // PB: Turn input off in manual mode
   END_STRUCT;
END_TYPE

// folder: Library Data Types/Devices/Status

TYPE "udtStatus_DigitalInput"
   STRUCT
      bOn : Bool;   // Digital Input is On
      bRisingEdge : Bool;   // Digital Input Rising Edge (TRUE for one-scan per edge)
      bFallingEdge : Bool;   // Digital Input Falling Edge (TRUE for one-scan per edge)
   END_STRUCT;
END_TYPE

TYPE "udtStatus_AnalogInput"
   STRUCT
      rCurrentValue : Real;   // Current analog input value in scaled engineering units
      bLowLow : Bool;   // Low low alarm is active
      bLow : Bool;   // Low warning is active
      bHigh : Bool;   // High warning is active
      bHighHigh : Bool;   // High high alarm is active
      bError : Bool;   // Error State Active
   END_STRUCT;
END_TYPE

TYPE "udtStatus_SolenoidValve"
   STRUCT
      bAtHome : Bool;   // Valve Home Feedback is Active
      bAtWork : Bool;   // Valve Work Feedback is Active
      bError : Bool;   // Valve Error State
   END_STRUCT;
END_TYPE

// folder: 5 - LIBRARY/Devices

FUNCTION_BLOCK "fbSolenoidValve"   // FB110, LAD
TITLE = Controls a double- or single-acting valve
{ S7_Optimized_Access := 'TRUE' }
VERSION : 0.1
   VAR_INPUT
      tInTimeout : Time;   // Timeout time for an actuator's feedback to activate before giving a fault
      iInMode : Int;   // Mode Selection
      bInEstop : Bool;   // Estop
      bInSignalHome : Bool;   // Home position feedback
      bInSignalWork : Bool;   // Work position feedback
      bInEnable : Bool;   // Home and Work Enabled
      bInCommandWork : Bool;   // Move to work position in automatic mode
      bInResetError : Bool;   // Reset Error
   END_VAR
   VAR_OUTPUT
      bOutCommandHome : Bool;   // Home position command
      bOutCommandWork : Bool;   // Work position command
      OutStatus : "udtStatus_SolenoidValve";   // Solenoid Valve Device Status
      ERROR_Valve : "udtError_SolenoidValve";   // Valve error structure
   END_VAR
   VAR_IN_OUT
      HMI_ValveControl : "udtHMI_SolenoidValve";   // HMI valve control
   END_VAR
   VAR
      ErrorScroller : "fbErrorScroller";   // Sub-block to handle error scroller
      TON_TimeOut : TON_TIME;   // Timer for Error Timeout
      Mode : Struct   // Device Mode
         iLast : Int;   // Last mode code
         bDidChange : Bool;   // New mode selected
         bAuto : Bool;   // Auto Mode is active
         bManual : Bool;   // Manual Mode is active
      END_STRUCT;
      PB : Struct   // HMI Control Pushbuttons
         bHome : Bool;   // Command device home in manual
         bWork : Bool;   // Command device work in manual
         bResetError : Bool;   // Reset errors
      END_STRUCT;
      bEnableHome : Bool;   // Home position enabled
      bEnableWork : Bool;   // Work position enabled
      bReset : Bool;   // Reset errors and timeout timer
      bTON_TimeOut : Bool;   // Timeout timer complete
   END_VAR
   VAR_TEMP   // added for the SCL form of the ladder/FBD networks
      _w1 : Bool;
   END_VAR
BEGIN

REGION Network 1: --------------------------------------------------------- Inputs ------------------------------------------------------------------
END_REGION

REGION Network 2: HMI Pushbutton: Command Home
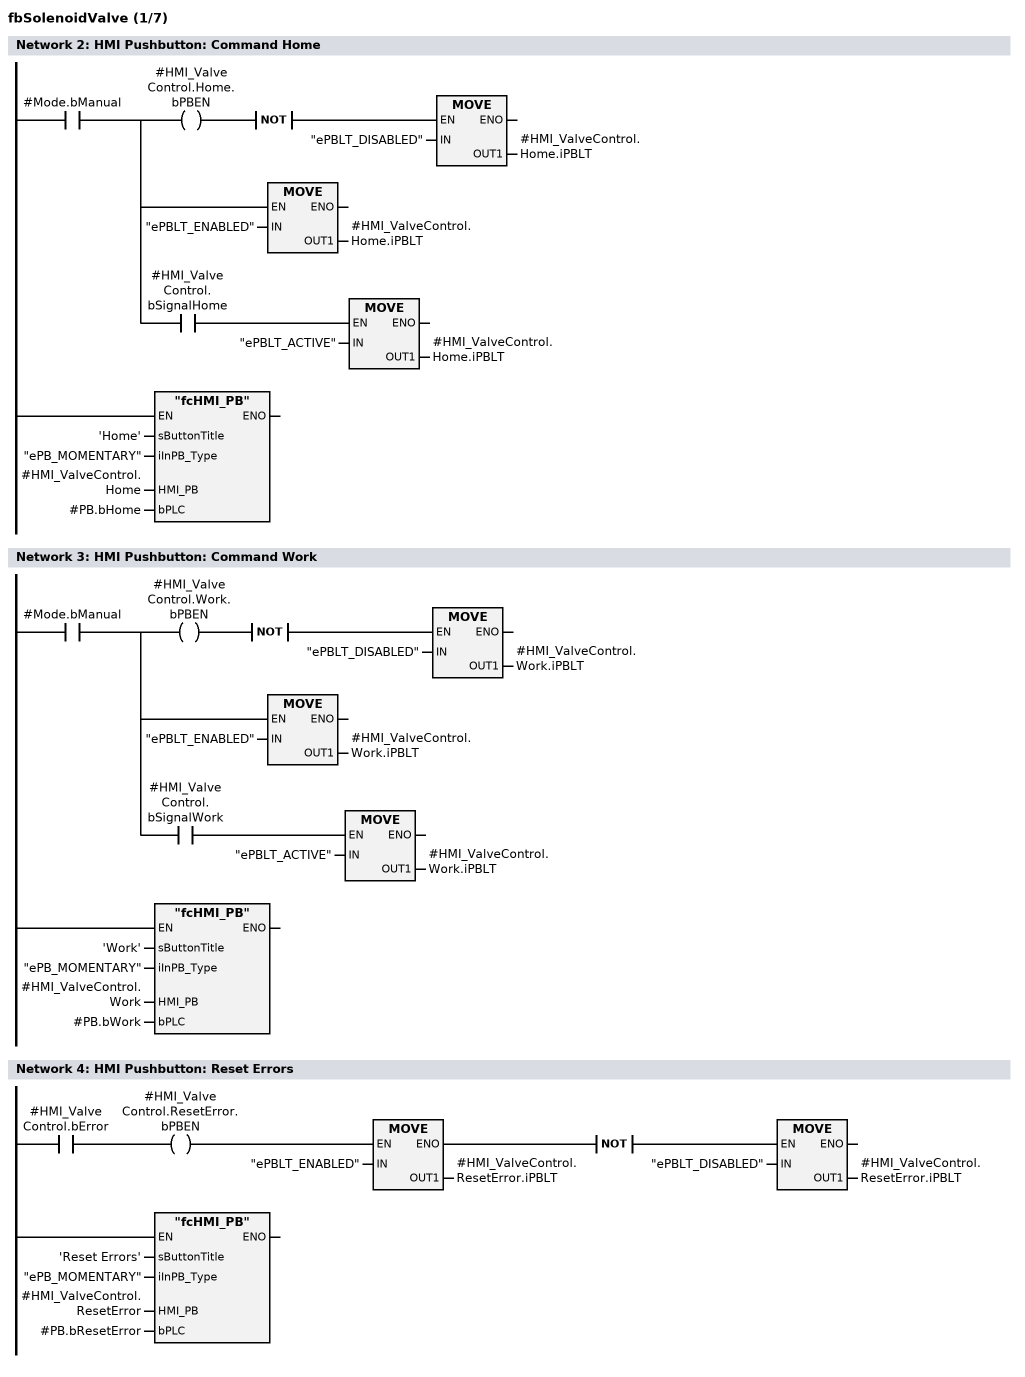
   RUNG wire#powerrail
      Contact( #Mode.bManual )
      wire#w1
      Coil( #HMI_ValveControl.Home.bPBEN )
      Not()
      Move(in := "ePBLT_DISABLED", out1 => #HMI_ValveControl.Home.iPBLT)
   END_RUNG
   RUNG wire#w1
      Move(in := "ePBLT_ENABLED", out1 => #HMI_ValveControl.Home.iPBLT)
   END_RUNG
   RUNG wire#w1
      Contact( #HMI_ValveControl.bSignalHome )
      Move(in := "ePBLT_ACTIVE", out1 => #HMI_ValveControl.Home.iPBLT)
   END_RUNG
   RUNG wire#powerrail
      "fcHMI_PB"(sButtonTitle := 'Home', iInPB_Type := "ePB_MOMENTARY", HMI_PB := #HMI_ValveControl.Home, bPLC := #PB.bHome)
   END_RUNG
   // the same network as SCL:
   #HMI_ValveControl.Home.bPBEN := #Mode.bManual;
   IF NOT #Mode.bManual THEN #HMI_ValveControl.Home.iPBLT := "ePBLT_DISABLED"; END_IF;
   IF #Mode.bManual THEN #HMI_ValveControl.Home.iPBLT := "ePBLT_ENABLED"; END_IF;
   IF #Mode.bManual AND #HMI_ValveControl.bSignalHome THEN
       #HMI_ValveControl.Home.iPBLT := "ePBLT_ACTIVE";
   END_IF;
   "fcHMI_PB"(sButtonTitle := 'Home',
              iInPB_Type := "ePB_MOMENTARY",
              HMI_PB := #HMI_ValveControl.Home,
              bPLC := #PB.bHome);
END_REGION

REGION Network 3: HMI Pushbutton: Command Work
   RUNG wire#powerrail
      Contact( #Mode.bManual )
      wire#w1
      Coil( #HMI_ValveControl.Work.bPBEN )
      Not()
      Move(in := "ePBLT_DISABLED", out1 => #HMI_ValveControl.Work.iPBLT)
   END_RUNG
   RUNG wire#w1
      Move(in := "ePBLT_ENABLED", out1 => #HMI_ValveControl.Work.iPBLT)
   END_RUNG
   RUNG wire#w1
      Contact( #HMI_ValveControl.bSignalWork )
      Move(in := "ePBLT_ACTIVE", out1 => #HMI_ValveControl.Work.iPBLT)
   END_RUNG
   RUNG wire#powerrail
      "fcHMI_PB"(sButtonTitle := 'Work', iInPB_Type := "ePB_MOMENTARY", HMI_PB := #HMI_ValveControl.Work, bPLC := #PB.bWork)
   END_RUNG
   // the same network as SCL:
   #HMI_ValveControl.Work.bPBEN := #Mode.bManual;
   IF NOT #Mode.bManual THEN #HMI_ValveControl.Work.iPBLT := "ePBLT_DISABLED"; END_IF;
   IF #Mode.bManual THEN #HMI_ValveControl.Work.iPBLT := "ePBLT_ENABLED"; END_IF;
   IF #Mode.bManual AND #HMI_ValveControl.bSignalWork THEN
       #HMI_ValveControl.Work.iPBLT := "ePBLT_ACTIVE";
   END_IF;
   "fcHMI_PB"(sButtonTitle := 'Work',
              iInPB_Type := "ePB_MOMENTARY",
              HMI_PB := #HMI_ValveControl.Work,
              bPLC := #PB.bWork);
END_REGION

REGION Network 4: HMI Pushbutton: Reset Errors
   RUNG wire#powerrail
      Contact( #HMI_ValveControl.bError )
      Coil( #HMI_ValveControl.ResetError.bPBEN )
      Move(in := "ePBLT_ENABLED", out1 => #HMI_ValveControl.ResetError.iPBLT)
      Not()
      Move(in := "ePBLT_DISABLED", out1 => #HMI_ValveControl.ResetError.iPBLT)
   END_RUNG
   RUNG wire#powerrail
      "fcHMI_PB"(sButtonTitle := 'Reset Errors', iInPB_Type := "ePB_MOMENTARY", HMI_PB := #HMI_ValveControl.ResetError, bPLC := #PB.bResetError)
   END_RUNG
   // the same network as SCL:
   #HMI_ValveControl.ResetError.bPBEN := #HMI_ValveControl.bError;
   IF #HMI_ValveControl.bError THEN #HMI_ValveControl.ResetError.iPBLT := "ePBLT_ENABLED"; END_IF;
   IF NOT #HMI_ValveControl.bError THEN #HMI_ValveControl.ResetError.iPBLT := "ePBLT_DISABLED"; END_IF;
   "fcHMI_PB"(sButtonTitle := 'Reset Errors',
              iInPB_Type := "ePB_MOMENTARY",
              HMI_PB := #HMI_ValveControl.ResetError,
              bPLC := #PB.bResetError);
END_REGION

REGION Network 5: Update the signal home bit
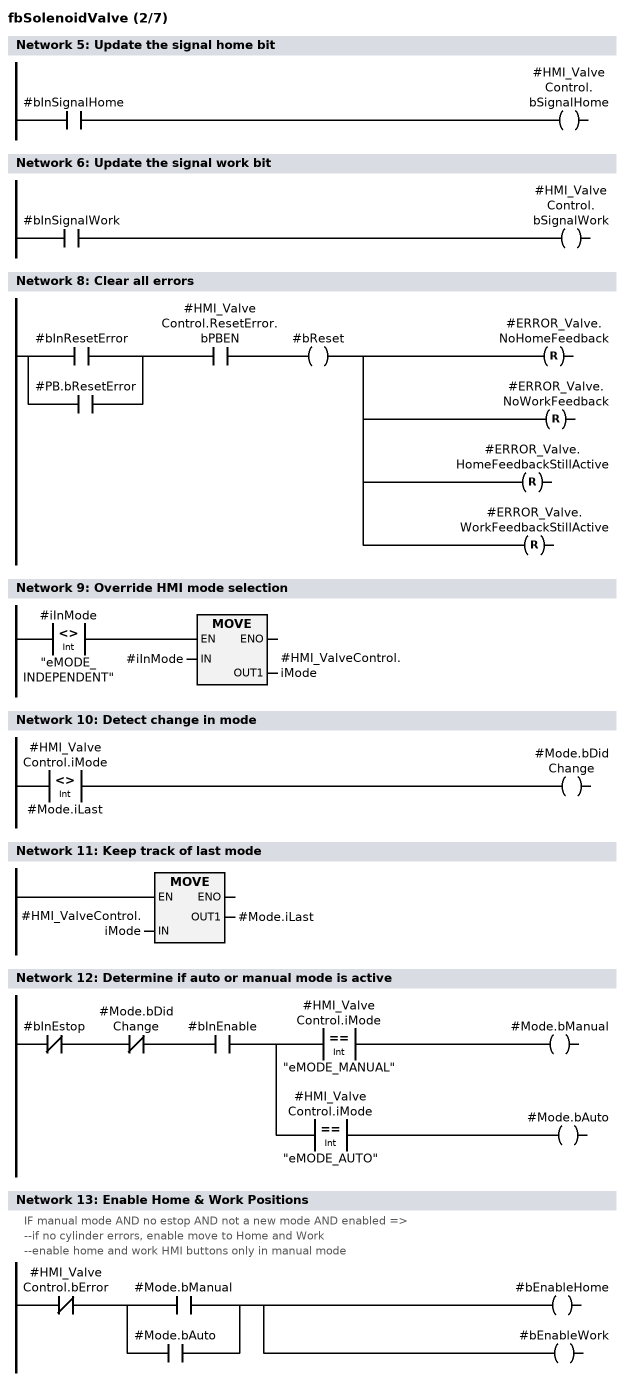
   RUNG wire#powerrail
      Contact( #bInSignalHome )
      Coil( #HMI_ValveControl.bSignalHome )
   END_RUNG
   // the same network as SCL:
   #HMI_ValveControl.bSignalHome := #bInSignalHome;
END_REGION

REGION Network 6: Update the signal work bit
   RUNG wire#powerrail
      Contact( #bInSignalWork )
      Coil( #HMI_ValveControl.bSignalWork )
   END_RUNG
   // the same network as SCL:
   #HMI_ValveControl.bSignalWork := #bInSignalWork;
END_REGION

REGION Network 7: --------------------------------------------------- Control Logic ------------------------------------------------------------
END_REGION

REGION Network 8: Clear all errors
   RUNG wire#powerrail
      Contact( #bInResetError )
      wire#w1
      Contact( #HMI_ValveControl.ResetError.bPBEN )
      Coil( #bReset )
      wire#w2
      R_Coil( #ERROR_Valve.NoHomeFeedback )
   END_RUNG
   RUNG wire#powerrail
      Contact( #PB.bResetError )
   END_RUNG wire#w1
   RUNG wire#w2
      R_Coil( #ERROR_Valve.NoWorkFeedback )
   END_RUNG
   RUNG wire#w2
      R_Coil( #ERROR_Valve.HomeFeedbackStillActive )
   END_RUNG
   RUNG wire#w2
      R_Coil( #ERROR_Valve.WorkFeedbackStillActive )
   END_RUNG
   // the same network as SCL:
   #bReset := (#bInResetError OR #PB.bResetError) AND #HMI_ValveControl.ResetError.bPBEN;
   IF #bReset THEN
       #ERROR_Valve.NoHomeFeedback := FALSE;
       #ERROR_Valve.NoWorkFeedback := FALSE;
       #ERROR_Valve.HomeFeedbackStillActive := FALSE;
       #ERROR_Valve.WorkFeedbackStillActive := FALSE;
   END_IF;
END_REGION

REGION Network 9: Override HMI mode selection
   RUNG wire#powerrail
      { S7_Templates := "SrcType := Int" } NE_Contact(in1 := #iInMode, in2 := "eMODE_INDEPENDENT")
      Move(in := #iInMode, out1 => #HMI_ValveControl.iMode)
   END_RUNG
   // the same network as SCL:
   IF #iInMode <> "eMODE_INDEPENDENT" THEN #HMI_ValveControl.iMode := #iInMode; END_IF;
END_REGION

REGION Network 10: Detect change in mode
   RUNG wire#powerrail
      { S7_Templates := "SrcType := Int" } NE_Contact(in1 := #HMI_ValveControl.iMode, in2 := #Mode.iLast)
      Coil( #Mode.bDidChange )
   END_RUNG
   // the same network as SCL:
   #Mode.bDidChange := #HMI_ValveControl.iMode <> #Mode.iLast;
END_REGION

REGION Network 11: Keep track of last mode
   RUNG wire#powerrail
      Move(in := #HMI_ValveControl.iMode, out1 => #Mode.iLast)
   END_RUNG
   // the same network as SCL:
   #Mode.iLast := #HMI_ValveControl.iMode;
END_REGION

REGION Network 12: Determine if auto or manual mode is active
   RUNG wire#powerrail
      I_Contact( #bInEstop )
      I_Contact( #Mode.bDidChange )
      Contact( #bInEnable )
      wire#w1
      { S7_Templates := "SrcType := Int" } EQ_Contact(in1 := #HMI_ValveControl.iMode, in2 := "eMODE_MANUAL")
      Coil( #Mode.bManual )
   END_RUNG
   RUNG wire#w1
      { S7_Templates := "SrcType := Int" } EQ_Contact(in1 := #HMI_ValveControl.iMode, in2 := "eMODE_AUTO")
      Coil( #Mode.bAuto )
   END_RUNG
   // the same network as SCL:
   #_w1 := NOT #bInEstop AND NOT #Mode.bDidChange AND #bInEnable;
   #Mode.bManual := #_w1 AND (#HMI_ValveControl.iMode = "eMODE_MANUAL");
   #Mode.bAuto := #_w1 AND (#HMI_ValveControl.iMode = "eMODE_AUTO");
END_REGION

REGION Network 13: Enable Home & Work Positions
   // IF manual mode AND no estop AND not a new mode AND enabled => 
   // --if no cylinder errors, enable move to Home and Work
   // --enable home and work HMI buttons only in manual mode
   RUNG wire#powerrail
      I_Contact( #HMI_ValveControl.bError )
      wire#w1
      Contact( #Mode.bManual )
      wire#w2
      Coil( #bEnableHome )
   END_RUNG
   RUNG wire#w1
      Contact( #Mode.bAuto )
   END_RUNG wire#w2
   RUNG wire#w2
      Coil( #bEnableWork )
   END_RUNG
   // the same network as SCL:
   #bEnableHome := NOT #HMI_ValveControl.bError AND (#Mode.bManual OR #Mode.bAuto);
   #bEnableWork := #bEnableHome;
END_REGION

REGION Network 14: Move to Home Position (Retracted)
   // IF manual mode and home button is pressed =>
   // --Set close cylinder
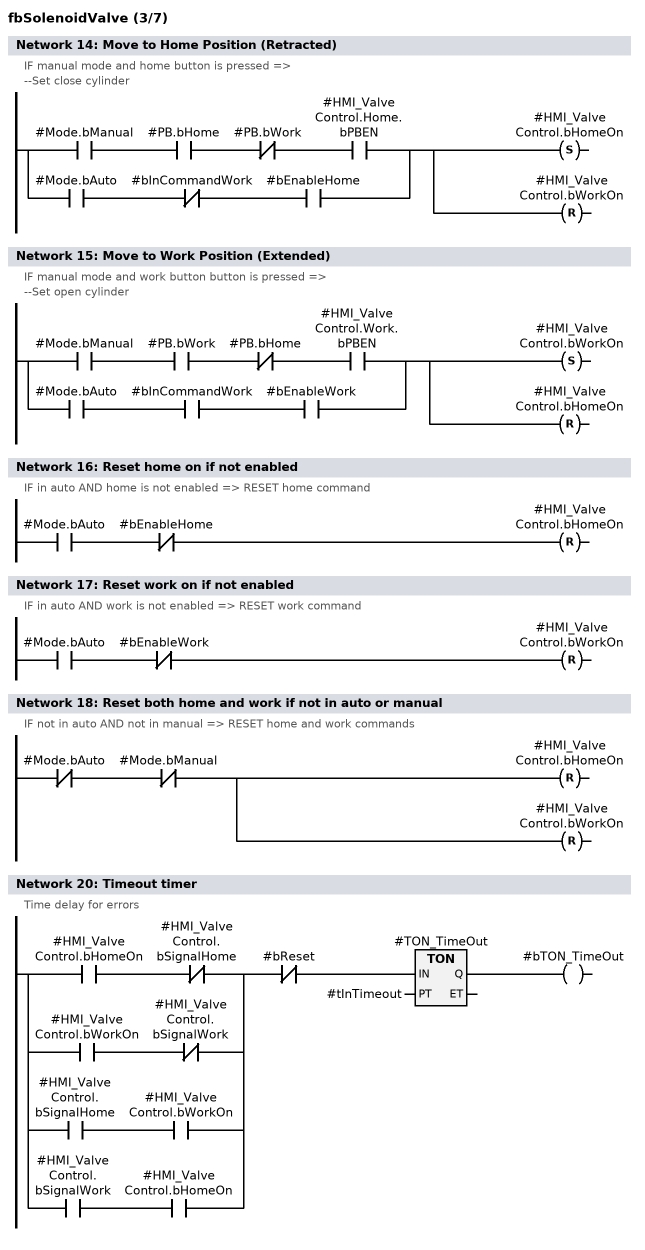
   RUNG wire#powerrail
      Contact( #Mode.bManual )
      Contact( #PB.bHome )
      I_Contact( #PB.bWork )
      Contact( #HMI_ValveControl.Home.bPBEN )
      wire#w1
      S_Coil( #HMI_ValveControl.bHomeOn )
   END_RUNG
   RUNG wire#powerrail
      Contact( #Mode.bAuto )
      I_Contact( #bInCommandWork )
      Contact( #bEnableHome )
   END_RUNG wire#w1
   RUNG wire#w1
      R_Coil( #HMI_ValveControl.bWorkOn )
   END_RUNG
   // the same network as SCL:
   IF (#Mode.bManual AND #PB.bHome AND NOT #PB.bWork AND #HMI_ValveControl.Home.bPBEN) OR (#Mode.bAuto AND NOT #bInCommandWork AND #bEnableHome) THEN
       #HMI_ValveControl.bHomeOn := TRUE;
       #HMI_ValveControl.bWorkOn := FALSE;
   END_IF;
END_REGION

REGION Network 15: Move to Work Position (Extended)
   // IF manual mode and work button button is pressed =>
   // --Set open cylinder
   RUNG wire#powerrail
      Contact( #Mode.bManual )
      Contact( #PB.bWork )
      I_Contact( #PB.bHome )
      Contact( #HMI_ValveControl.Work.bPBEN )
      wire#w1
      S_Coil( #HMI_ValveControl.bWorkOn )
   END_RUNG
   RUNG wire#powerrail
      Contact( #Mode.bAuto )
      Contact( #bInCommandWork )
      Contact( #bEnableWork )
   END_RUNG wire#w1
   RUNG wire#w1
      R_Coil( #HMI_ValveControl.bHomeOn )
   END_RUNG
   // the same network as SCL:
   IF (#Mode.bManual AND #PB.bWork AND NOT #PB.bHome AND #HMI_ValveControl.Work.bPBEN) OR (#Mode.bAuto AND #bInCommandWork AND #bEnableWork) THEN
       #HMI_ValveControl.bWorkOn := TRUE;
       #HMI_ValveControl.bHomeOn := FALSE;
   END_IF;
END_REGION

REGION Network 16: Reset home on if not enabled
   // IF in auto AND home is not enabled => RESET home command
   RUNG wire#powerrail
      Contact( #Mode.bAuto )
      I_Contact( #bEnableHome )
      R_Coil( #HMI_ValveControl.bHomeOn )
   END_RUNG
   // the same network as SCL:
   IF #Mode.bAuto AND NOT #bEnableHome THEN #HMI_ValveControl.bHomeOn := FALSE; END_IF;
END_REGION

REGION Network 17: Reset work on if not enabled
   // IF in auto AND work is not enabled => RESET work command
   RUNG wire#powerrail
      Contact( #Mode.bAuto )
      I_Contact( #bEnableWork )
      R_Coil( #HMI_ValveControl.bWorkOn )
   END_RUNG
   // the same network as SCL:
   IF #Mode.bAuto AND NOT #bEnableWork THEN #HMI_ValveControl.bWorkOn := FALSE; END_IF;
END_REGION

REGION Network 18: Reset both home and work if not in auto or manual
   // IF not in auto AND not in manual => RESET home and work commands
   RUNG wire#powerrail
      I_Contact( #Mode.bAuto )
      I_Contact( #Mode.bManual )
      wire#w1
      R_Coil( #HMI_ValveControl.bHomeOn )
   END_RUNG
   RUNG wire#w1
      R_Coil( #HMI_ValveControl.bWorkOn )
   END_RUNG
   // the same network as SCL:
   IF NOT #Mode.bAuto AND NOT #Mode.bManual THEN
       #HMI_ValveControl.bHomeOn := FALSE;
       #HMI_ValveControl.bWorkOn := FALSE;
   END_IF;
END_REGION

REGION Network 19: --------------------------------------------------------- Errors ------------------------------------------------------------------
END_REGION

REGION Network 20: Timeout timer
   // Time delay for errors
   #TON_TimeOut(IN := ((#HMI_ValveControl.bHomeOn AND NOT #HMI_ValveControl.bSignalHome) OR (#HMI_ValveControl.bWorkOn AND NOT #HMI_ValveControl.bSignalWork) OR (#HMI_ValveControl.bSignalHome AND #HMI_ValveControl.bWorkOn) OR (#HMI_ValveControl.bSignalWork AND #HMI_ValveControl.bHomeOn)) AND NOT #bReset,   // TON
                PT := #tInTimeout);
   #bTON_TimeOut := #TON_TimeOut.Q;
END_REGION

REGION Network 21: Error: Home position feedback not active
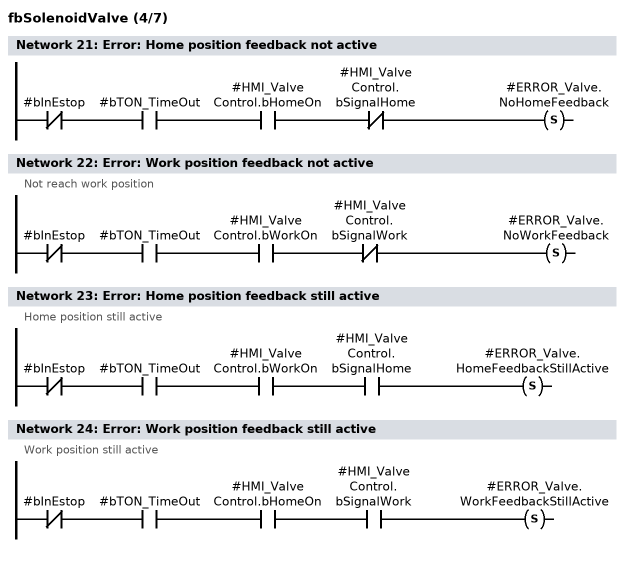
   RUNG wire#powerrail
      I_Contact( #bInEstop )
      Contact( #bTON_TimeOut )
      Contact( #HMI_ValveControl.bHomeOn )
      I_Contact( #HMI_ValveControl.bSignalHome )
      S_Coil( #ERROR_Valve.NoHomeFeedback )
   END_RUNG
   // the same network as SCL:
   IF NOT #bInEstop AND #bTON_TimeOut AND #HMI_ValveControl.bHomeOn AND NOT #HMI_ValveControl.bSignalHome THEN
       #ERROR_Valve.NoHomeFeedback := TRUE;
   END_IF;
END_REGION

REGION Network 22: Error: Work position feedback not active
   // Not reach work position
   RUNG wire#powerrail
      I_Contact( #bInEstop )
      Contact( #bTON_TimeOut )
      Contact( #HMI_ValveControl.bWorkOn )
      I_Contact( #HMI_ValveControl.bSignalWork )
      S_Coil( #ERROR_Valve.NoWorkFeedback )
   END_RUNG
   // the same network as SCL:
   IF NOT #bInEstop AND #bTON_TimeOut AND #HMI_ValveControl.bWorkOn AND NOT #HMI_ValveControl.bSignalWork THEN
       #ERROR_Valve.NoWorkFeedback := TRUE;
   END_IF;
END_REGION

REGION Network 23: Error: Home position feedback still active
   // Home position still active
   RUNG wire#powerrail
      I_Contact( #bInEstop )
      Contact( #bTON_TimeOut )
      Contact( #HMI_ValveControl.bWorkOn )
      Contact( #HMI_ValveControl.bSignalHome )
      S_Coil( #ERROR_Valve.HomeFeedbackStillActive )
   END_RUNG
   // the same network as SCL:
   IF NOT #bInEstop AND #bTON_TimeOut AND #HMI_ValveControl.bWorkOn AND #HMI_ValveControl.bSignalHome THEN
       #ERROR_Valve.HomeFeedbackStillActive := TRUE;
   END_IF;
END_REGION

REGION Network 24: Error: Work position feedback still active
   // Work position still active
   RUNG wire#powerrail
      I_Contact( #bInEstop )
      Contact( #bTON_TimeOut )
      Contact( #HMI_ValveControl.bHomeOn )
      Contact( #HMI_ValveControl.bSignalWork )
      S_Coil( #ERROR_Valve.WorkFeedbackStillActive )
   END_RUNG
   // the same network as SCL:
   IF NOT #bInEstop AND #bTON_TimeOut AND #HMI_ValveControl.bHomeOn AND #HMI_ValveControl.bSignalWork THEN
       #ERROR_Valve.WorkFeedbackStillActive := TRUE;
   END_IF;
END_REGION

REGION Network 25: Error scroller
   // Call the Error-Scroller which cyles through all possible errors and checks 
   // their state for display on the HMI
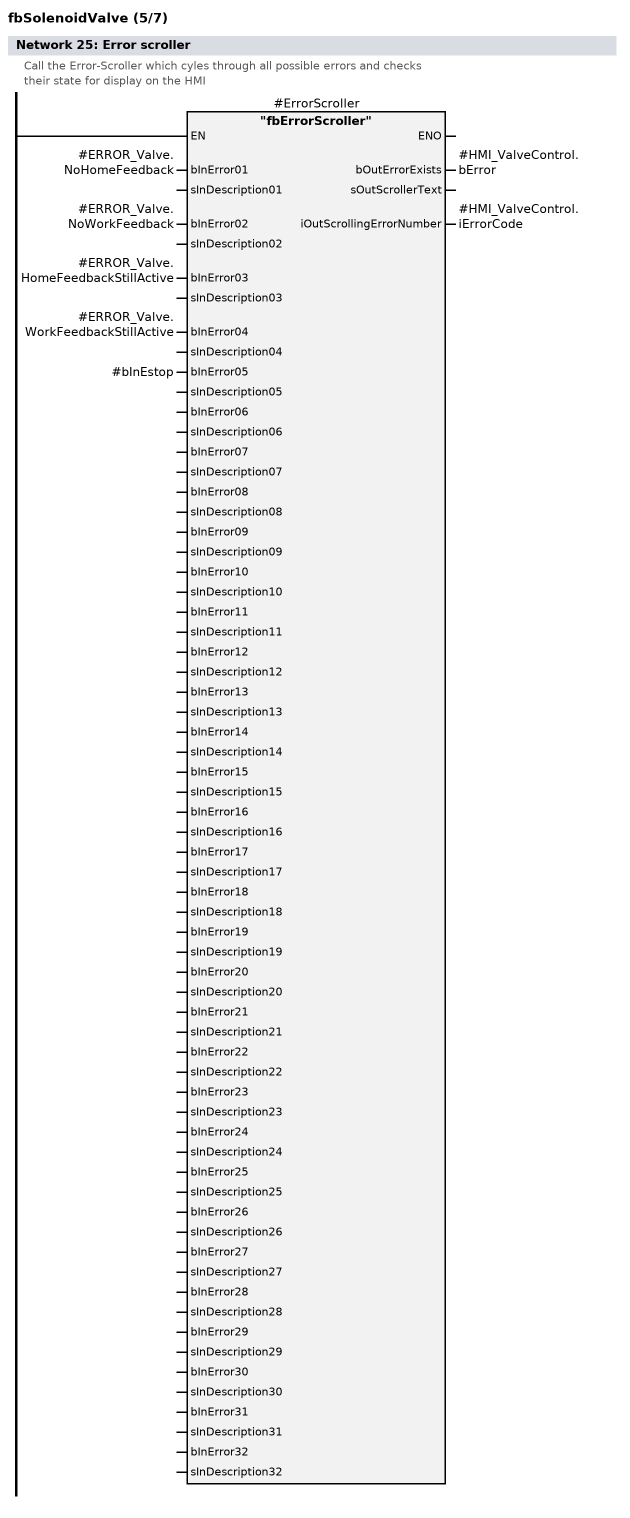
   RUNG wire#powerrail
      #ErrorScroller(bInError01 := #ERROR_Valve.NoHomeFeedback, sInDescription01 :=, bInError02 := #ERROR_Valve.NoWorkFeedback, sInDescription02 :=, bInError03 := #ERROR_Valve.HomeFeedbackStillActive, sInDescription03 :=, bInError04 := #ERROR_Valve.WorkFeedbackStillActive, sInDescription04 :=, bInError05 := #bInEstop, sInDescription05 :=, bInError06 :=, sInDescription06 :=, bInError07 :=, sInDescription07 :=, bInError08 :=, sInDescription08 :=, bInError09 :=, sInDescription09 :=, bInError10 :=, sInDescription10 :=, bInError11 :=, sInDescription11 :=, bInError12 :=, sInDescription12 :=, bInError13 :=, sInDescription13 :=, bInError14 :=, sInDescription14 :=, bInError15 :=, sInDescription15 :=, bInError16 :=, sInDescription16 :=, bInError17 :=, sInDescription17 :=, bInError18 :=, sInDescription18 :=, bInError19 :=, sInDescription19 :=, bInError20 :=, sInDescription20 :=, bInError21 :=, sInDescription21 :=, bInError22 :=, sInDescription22 :=, bInError23 :=, sInDescription23 :=, bInError24 :=, sInDescription24 :=, bInError25 :=, sInDescription25 :=, bInError26 :=, sInDescription26 :=, bInError27 :=, sInDescription27 :=, bInError28 :=, sInDescription28 :=, bInError29 :=, sInDescription29 :=, bInError30 :=, sInDescription30 :=, bInError31 :=, sInDescription31 :=, bInError32 :=, sInDescription32 :=, bOutErrorExists => #HMI_ValveControl.bError, sOutScrollerText =>, iOutScrollingErrorNumber => #HMI_ValveControl.iErrorCode)
   END_RUNG
   // the same network as SCL:
   #ErrorScroller(bInError01 := #ERROR_Valve.NoHomeFeedback,   // "fbErrorScroller"
                  bInError02 := #ERROR_Valve.NoWorkFeedback,
                  bInError03 := #ERROR_Valve.HomeFeedbackStillActive,
                  bInError04 := #ERROR_Valve.WorkFeedbackStillActive,
                  bInError05 := #bInEstop,
                  bOutErrorExists => #HMI_ValveControl.bError,
                  iOutScrollingErrorNumber => #HMI_ValveControl.iErrorCode);
END_REGION

REGION Network 26: Interlock
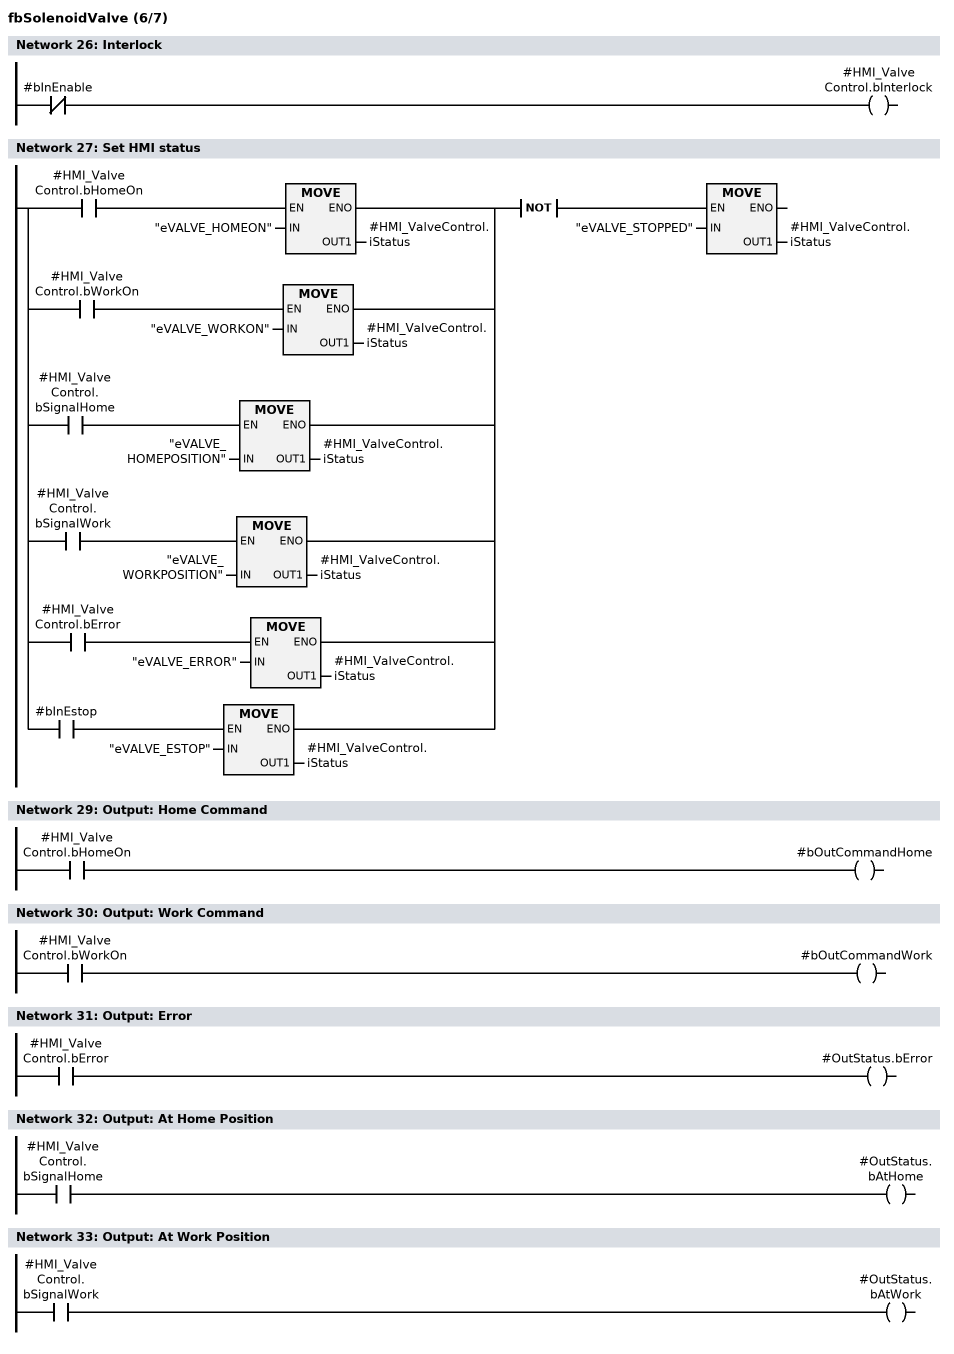
   RUNG wire#powerrail
      I_Contact( #bInEnable )
      Coil( #HMI_ValveControl.bInterlock )
   END_RUNG
   // the same network as SCL:
   #HMI_ValveControl.bInterlock := NOT #bInEnable;
END_REGION

REGION Network 27: Set HMI status
   RUNG wire#powerrail
      Contact( #HMI_ValveControl.bHomeOn )
      Move(in := "eVALVE_HOMEON", out1 => #HMI_ValveControl.iStatus)
      wire#w1
      Not()
      Move(in := "eVALVE_STOPPED", out1 => #HMI_ValveControl.iStatus)
   END_RUNG
   RUNG wire#powerrail
      Contact( #HMI_ValveControl.bWorkOn )
      Move(in := "eVALVE_WORKON", out1 => #HMI_ValveControl.iStatus)
   END_RUNG wire#w1
   RUNG wire#powerrail
      Contact( #HMI_ValveControl.bSignalHome )
      Move(in := "eVALVE_HOMEPOSITION", out1 => #HMI_ValveControl.iStatus)
   END_RUNG wire#w1
   RUNG wire#powerrail
      Contact( #HMI_ValveControl.bSignalWork )
      Move(in := "eVALVE_WORKPOSITION", out1 => #HMI_ValveControl.iStatus)
   END_RUNG wire#w1
   RUNG wire#powerrail
      Contact( #HMI_ValveControl.bError )
      Move(in := "eVALVE_ERROR", out1 => #HMI_ValveControl.iStatus)
   END_RUNG wire#w1
   RUNG wire#powerrail
      Contact( #bInEstop )
      Move(in := "eVALVE_ESTOP", out1 => #HMI_ValveControl.iStatus)
   END_RUNG wire#w1
   // the same network as SCL:
   IF #HMI_ValveControl.bHomeOn THEN #HMI_ValveControl.iStatus := "eVALVE_HOMEON"; END_IF;
   IF #HMI_ValveControl.bWorkOn THEN #HMI_ValveControl.iStatus := "eVALVE_WORKON"; END_IF;
   IF #HMI_ValveControl.bSignalHome THEN #HMI_ValveControl.iStatus := "eVALVE_HOMEPOSITION"; END_IF;
   IF #HMI_ValveControl.bSignalWork THEN #HMI_ValveControl.iStatus := "eVALVE_WORKPOSITION"; END_IF;
   IF #HMI_ValveControl.bError THEN #HMI_ValveControl.iStatus := "eVALVE_ERROR"; END_IF;
   IF #bInEstop THEN #HMI_ValveControl.iStatus := "eVALVE_ESTOP"; END_IF;
   IF NOT (#HMI_ValveControl.bHomeOn OR #HMI_ValveControl.bWorkOn OR #HMI_ValveControl.bSignalHome OR #HMI_ValveControl.bSignalWork OR #HMI_ValveControl.bError OR #bInEstop) THEN
       #HMI_ValveControl.iStatus := "eVALVE_STOPPED";
   END_IF;
END_REGION

REGION Network 28: -------------------------------------------------- Outputs --------------------------------------------------
END_REGION

REGION Network 29: Output: Home Command
   RUNG wire#powerrail
      Contact( #HMI_ValveControl.bHomeOn )
      Coil( #bOutCommandHome )
   END_RUNG
   // the same network as SCL:
   #bOutCommandHome := #HMI_ValveControl.bHomeOn;
END_REGION

REGION Network 30: Output: Work Command
   RUNG wire#powerrail
      Contact( #HMI_ValveControl.bWorkOn )
      Coil( #bOutCommandWork )
   END_RUNG
   // the same network as SCL:
   #bOutCommandWork := #HMI_ValveControl.bWorkOn;
END_REGION

REGION Network 31: Output: Error
   RUNG wire#powerrail
      Contact( #HMI_ValveControl.bError )
      Coil( #OutStatus.bError )
   END_RUNG
   // the same network as SCL:
   #OutStatus.bError := #HMI_ValveControl.bError;
END_REGION

REGION Network 32: Output: At Home Position
   RUNG wire#powerrail
      Contact( #HMI_ValveControl.bSignalHome )
      Coil( #OutStatus.bAtHome )
   END_RUNG
   // the same network as SCL:
   #OutStatus.bAtHome := #HMI_ValveControl.bSignalHome;
END_REGION

REGION Network 33: Output: At Work Position
   RUNG wire#powerrail
      Contact( #HMI_ValveControl.bSignalWork )
      Coil( #OutStatus.bAtWork )
   END_RUNG
   // the same network as SCL:
   #OutStatus.bAtWork := #HMI_ValveControl.bSignalWork;
END_REGION

REGION Network 34: Set ENO
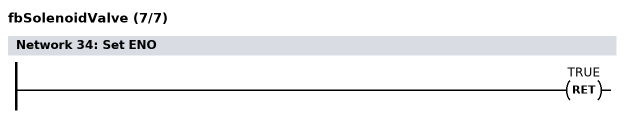
   RUNG wire#powerrail
      ReturnCoil( TRUE )
   END_RUNG
   // the same network as SCL:
   ENO := TRUE;
   RETURN;
END_REGION
END_FUNCTION_BLOCK

FUNCTION_BLOCK "fbAnalogInput"   // FB140, LAD
TITLE = Reads and controls an analog input
{ S7_Optimized_Access := 'TRUE' }
VERSION : 0.1
   VAR_INPUT
      iInMode : Int;   // Current mode
      wInValue : Word;   // Actual analog input value
      iInSensorType : Int;   // Enum of sensor types (IoScaling.S7Analog.Types)
      rInEngUnitsMin : Real;   // Engineering units scale min
      rInEngUnitsMax : Real;   // Engineering units scale max
      rInLowLow : Real := -3.402823E+38;   // Low low alarm set point
      rInLow : Real := -3.402823E+38;   // Low warning set point
      rInHigh : Real := 3.402823E+38;   // High warning set point
      rInHighHigh : Real := 3.402823E+38;   // High high alarm set point
      rInLowLowDeadband : Real := 0.0;   // Low low deadband amount
      rInLowDeadband : Real := 0.0;   // Low deadband amount
      rInHighDeadband : Real := 0.0;   // High deadband amount
      rInHighHighDeadband : Real := 0.0;   // High high deadband amount
      bInResetError : Bool;   // Reset block errors
   END_VAR
   VAR_OUTPUT
      OutStatus : "udtStatus_AnalogInput";   // Analog Input Device Status
      ERROR_IO_AnalogInput : "udtError_AnalogInput";   // Error structure for an analog input
   END_VAR
   VAR_IN_OUT
      HMI_IO_AnalogInput : "udtHMI_AnalogInput";   // HMI control structure for an analog input
   END_VAR
   VAR
      ErrorScroller : "fbErrorScroller";   // Scrolls errors on the HMI
      iRawMin : Int := 0;   // Raw input min value
      iRawMax : Int := 27648;   // Raw input max value
      rScaledMin : Real := 0.0;   // Scaled input min value
      rScaledMax : Real := 100.0;   // Scaled input max value
      bReset : Bool;   // Reset requested
      bScalingError : Bool;   // Error when scaling input
      PB : Struct
         bResetError : Bool;
      END_STRUCT;
   END_VAR
   VAR_TEMP
      bTemp : Bool;
      rTemp : Real;
   END_VAR
BEGIN

REGION Network 1: --------------------------------------------------------- Inputs ------------------------------------------------------------------
END_REGION

REGION Network 2: HMI Pushbutton: Reset Errors
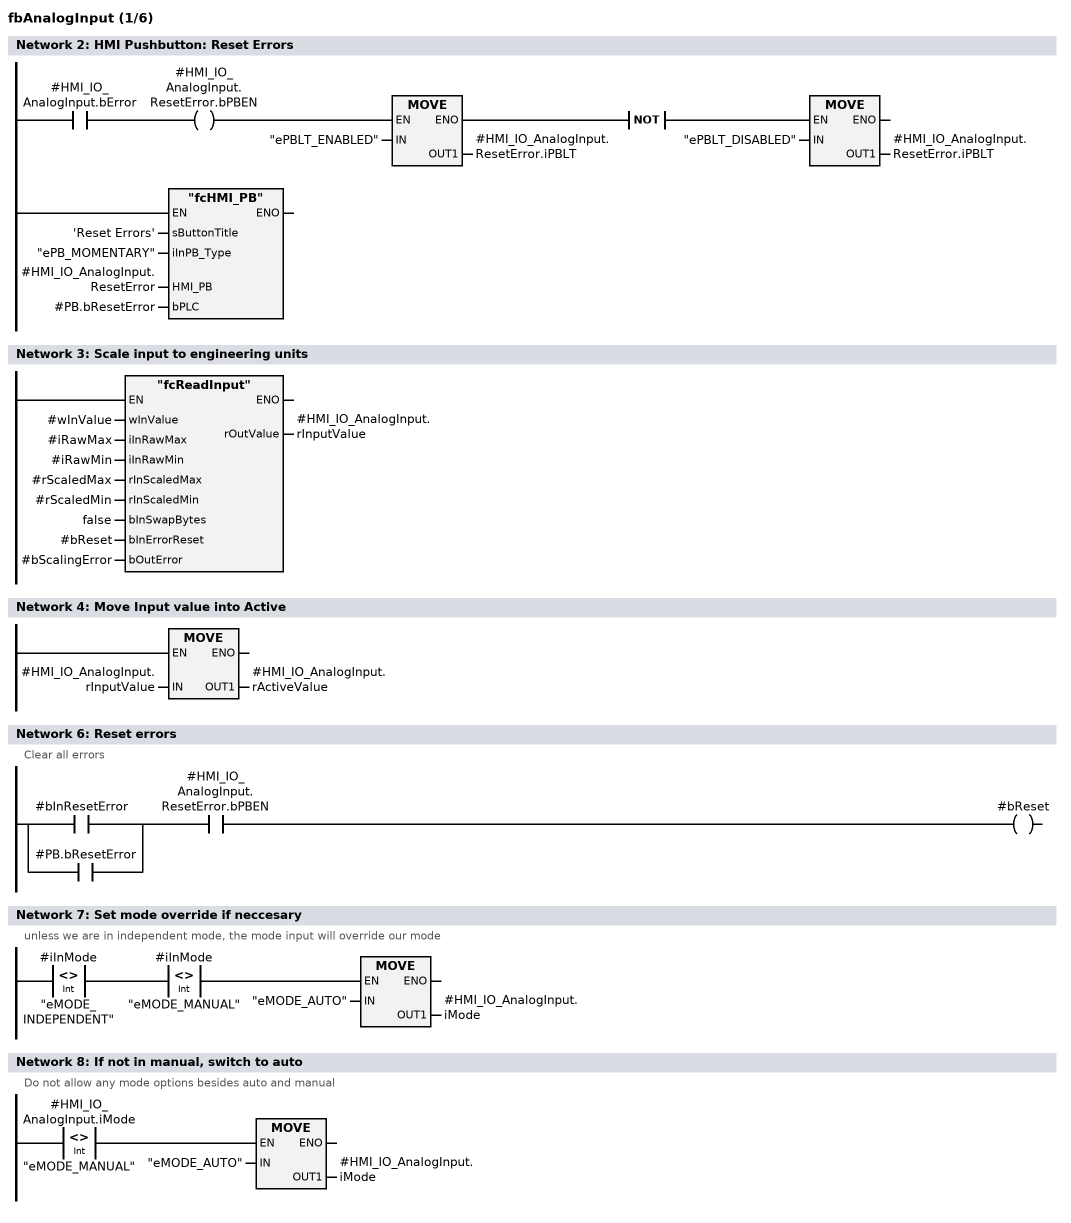
   RUNG wire#powerrail
      Contact( #HMI_IO_AnalogInput.bError )
      Coil( #HMI_IO_AnalogInput.ResetError.bPBEN )
      Move(in := "ePBLT_ENABLED", out1 => #HMI_IO_AnalogInput.ResetError.iPBLT)
      Not()
      Move(in := "ePBLT_DISABLED", out1 => #HMI_IO_AnalogInput.ResetError.iPBLT)
   END_RUNG
   RUNG wire#powerrail
      "fcHMI_PB"(sButtonTitle := 'Reset Errors', iInPB_Type := "ePB_MOMENTARY", HMI_PB := #HMI_IO_AnalogInput.ResetError, bPLC := #PB.bResetError)
   END_RUNG
   // the same network as SCL:
   #HMI_IO_AnalogInput.ResetError.bPBEN := #HMI_IO_AnalogInput.bError;
   IF #HMI_IO_AnalogInput.bError THEN #HMI_IO_AnalogInput.ResetError.iPBLT := "ePBLT_ENABLED"; END_IF;
   IF NOT #HMI_IO_AnalogInput.bError THEN #HMI_IO_AnalogInput.ResetError.iPBLT := "ePBLT_DISABLED"; END_IF;
   "fcHMI_PB"(sButtonTitle := 'Reset Errors',
              iInPB_Type := "ePB_MOMENTARY",
              HMI_PB := #HMI_IO_AnalogInput.ResetError,
              bPLC := #PB.bResetError);
END_REGION

REGION Network 3: Scale input to engineering units
   RUNG wire#powerrail
      "fcReadInput"(wInValue := #wInValue, iInRawMax := #iRawMax, iInRawMin := #iRawMin, rInScaledMax := #rScaledMax, rInScaledMin := #rScaledMin, bInSwapBytes := false, bInErrorReset := #bReset, bOutError := #bScalingError, rOutValue => #HMI_IO_AnalogInput.rInputValue)
   END_RUNG
   // the same network as SCL:
   "fcReadInput"(wInValue := #wInValue,
                 iInRawMax := #iRawMax,
                 iInRawMin := #iRawMin,
                 rInScaledMax := #rScaledMax,
                 rInScaledMin := #rScaledMin,
                 bInSwapBytes := false,
                 bInErrorReset := #bReset,
                 bOutError := #bScalingError,
                 rOutValue => #HMI_IO_AnalogInput.rInputValue);
END_REGION

REGION Network 4: Move Input value into Active
   RUNG wire#powerrail
      Move(in := #HMI_IO_AnalogInput.rInputValue, out1 => #HMI_IO_AnalogInput.rActiveValue)
   END_RUNG
   // the same network as SCL:
   #HMI_IO_AnalogInput.rActiveValue := #HMI_IO_AnalogInput.rInputValue;
END_REGION

REGION Network 5: --------------------------------------------------- Control Logic ------------------------------------------------------------
END_REGION

REGION Network 6: Reset errors
   // Clear all errors
   RUNG wire#powerrail
      Contact( #bInResetError )
      wire#w1
      Contact( #HMI_IO_AnalogInput.ResetError.bPBEN )
      Coil( #bReset )
   END_RUNG
   RUNG wire#powerrail
      Contact( #PB.bResetError )
   END_RUNG wire#w1
   // the same network as SCL:
   #bReset := (#bInResetError OR #PB.bResetError) AND #HMI_IO_AnalogInput.ResetError.bPBEN;
END_REGION

REGION Network 7: Set mode override if neccesary
   // unless we are in independent mode, the mode input will override our mode
   RUNG wire#powerrail
      { S7_Templates := "SrcType := Int" } NE_Contact(in1 := #iInMode, in2 := "eMODE_INDEPENDENT")
      { S7_Templates := "SrcType := Int" } NE_Contact(in1 := #iInMode, in2 := "eMODE_MANUAL")
      Move(in := "eMODE_AUTO", out1 => #HMI_IO_AnalogInput.iMode)
   END_RUNG
   // the same network as SCL:
   IF (#iInMode <> "eMODE_INDEPENDENT") AND (#iInMode <> "eMODE_MANUAL") THEN
       #HMI_IO_AnalogInput.iMode := "eMODE_AUTO";
   END_IF;
END_REGION

REGION Network 8: If not in manual, switch to auto
   // Do not allow any mode options besides auto and manual
   RUNG wire#powerrail
      { S7_Templates := "SrcType := Int" } NE_Contact(in1 := #HMI_IO_AnalogInput.iMode, in2 := "eMODE_MANUAL")
      Move(in := "eMODE_AUTO", out1 => #HMI_IO_AnalogInput.iMode)
   END_RUNG
   // the same network as SCL:
   IF #HMI_IO_AnalogInput.iMode <> "eMODE_MANUAL" THEN #HMI_IO_AnalogInput.iMode := "eMODE_AUTO"; END_IF;
END_REGION

REGION Network 9: Determine if manual mode is active
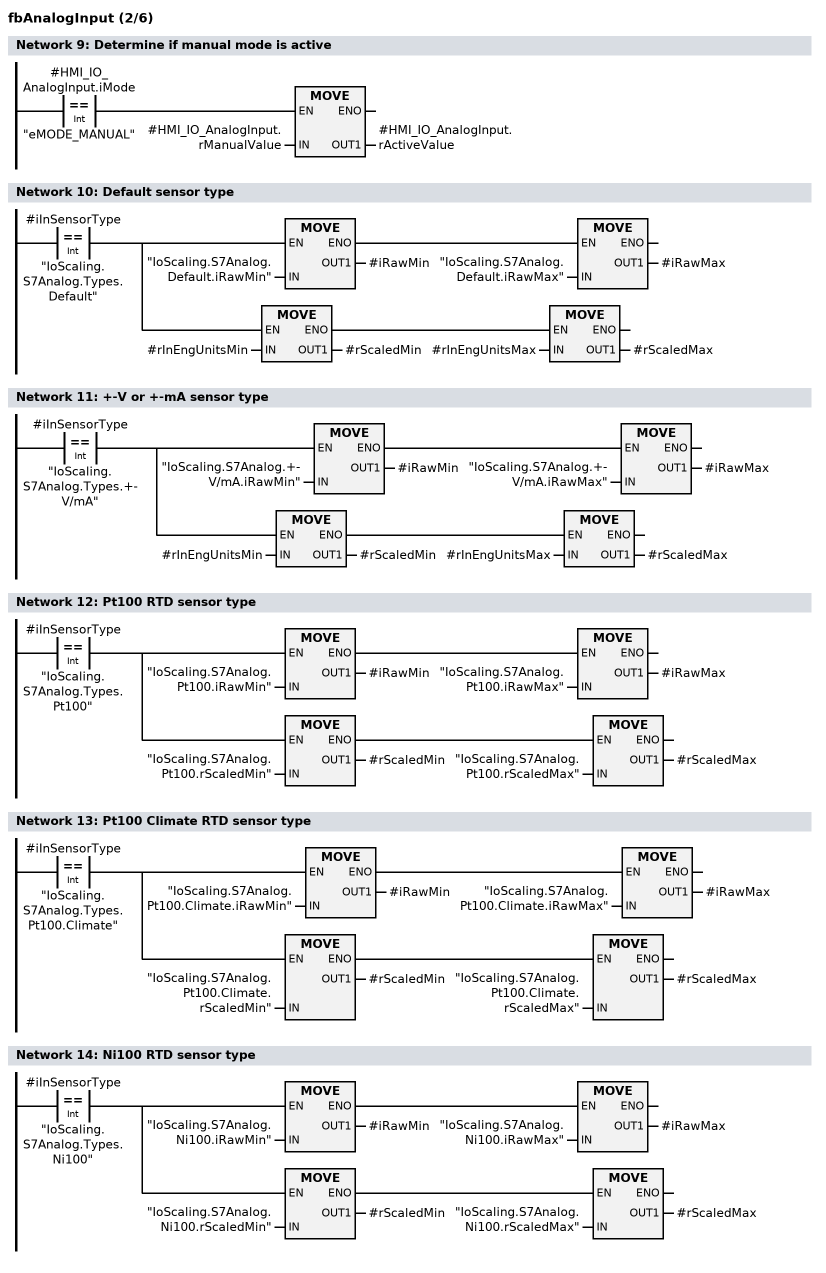
   RUNG wire#powerrail
      { S7_Templates := "SrcType := Int" } EQ_Contact(in1 := #HMI_IO_AnalogInput.iMode, in2 := "eMODE_MANUAL")
      Move(in := #HMI_IO_AnalogInput.rManualValue, out1 => #HMI_IO_AnalogInput.rActiveValue)
   END_RUNG
   // the same network as SCL:
   IF #HMI_IO_AnalogInput.iMode = "eMODE_MANUAL" THEN
       #HMI_IO_AnalogInput.rActiveValue := #HMI_IO_AnalogInput.rManualValue;
   END_IF;
END_REGION

REGION Network 10: Default sensor type
   RUNG wire#powerrail
      { S7_Templates := "SrcType := Int" } EQ_Contact(in1 := #iInSensorType, in2 := "IoScaling.S7Analog.Types.Default")
      wire#w1
      Move(in := "IoScaling.S7Analog.Default.iRawMin", out1 => #iRawMin)
      Move(in := "IoScaling.S7Analog.Default.iRawMax", out1 => #iRawMax)
   END_RUNG
   RUNG wire#w1
      Move(in := #rInEngUnitsMin, out1 => #rScaledMin)
      Move(in := #rInEngUnitsMax, out1 => #rScaledMax)
   END_RUNG
   // the same network as SCL:
   IF #iInSensorType = "IoScaling.S7Analog.Types.Default" THEN
       #iRawMin := "IoScaling.S7Analog.Default.iRawMin";
       #iRawMax := "IoScaling.S7Analog.Default.iRawMax";
       #rScaledMin := #rInEngUnitsMin;
       #rScaledMax := #rInEngUnitsMax;
   END_IF;
END_REGION

REGION Network 11: +-V or +-mA sensor type
   RUNG wire#powerrail
      { S7_Templates := "SrcType := Int" } EQ_Contact(in1 := #iInSensorType, in2 := "IoScaling.S7Analog.Types.+-V/mA")
      wire#w1
      Move(in := "IoScaling.S7Analog.+-V/mA.iRawMin", out1 => #iRawMin)
      Move(in := "IoScaling.S7Analog.+-V/mA.iRawMax", out1 => #iRawMax)
   END_RUNG
   RUNG wire#w1
      Move(in := #rInEngUnitsMin, out1 => #rScaledMin)
      Move(in := #rInEngUnitsMax, out1 => #rScaledMax)
   END_RUNG
   // the same network as SCL:
   IF #iInSensorType = "IoScaling.S7Analog.Types.+-V/mA" THEN
       #iRawMin := "IoScaling.S7Analog.+-V/mA.iRawMin";
       #iRawMax := "IoScaling.S7Analog.+-V/mA.iRawMax";
       #rScaledMin := #rInEngUnitsMin;
       #rScaledMax := #rInEngUnitsMax;
   END_IF;
END_REGION

REGION Network 12: Pt100 RTD sensor type
   RUNG wire#powerrail
      { S7_Templates := "SrcType := Int" } EQ_Contact(in1 := #iInSensorType, in2 := "IoScaling.S7Analog.Types.Pt100")
      wire#w1
      Move(in := "IoScaling.S7Analog.Pt100.iRawMin", out1 => #iRawMin)
      Move(in := "IoScaling.S7Analog.Pt100.iRawMax", out1 => #iRawMax)
   END_RUNG
   RUNG wire#w1
      Move(in := "IoScaling.S7Analog.Pt100.rScaledMin", out1 => #rScaledMin)
      Move(in := "IoScaling.S7Analog.Pt100.rScaledMax", out1 => #rScaledMax)
   END_RUNG
   // the same network as SCL:
   IF #iInSensorType = "IoScaling.S7Analog.Types.Pt100" THEN
       #iRawMin := "IoScaling.S7Analog.Pt100.iRawMin";
       #iRawMax := "IoScaling.S7Analog.Pt100.iRawMax";
       #rScaledMin := "IoScaling.S7Analog.Pt100.rScaledMin";
       #rScaledMax := "IoScaling.S7Analog.Pt100.rScaledMax";
   END_IF;
END_REGION

REGION Network 13: Pt100 Climate RTD sensor type
   RUNG wire#powerrail
      { S7_Templates := "SrcType := Int" } EQ_Contact(in1 := #iInSensorType, in2 := "IoScaling.S7Analog.Types.Pt100.Climate")
      wire#w1
      Move(in := "IoScaling.S7Analog.Pt100.Climate.iRawMin", out1 => #iRawMin)
      Move(in := "IoScaling.S7Analog.Pt100.Climate.iRawMax", out1 => #iRawMax)
   END_RUNG
   RUNG wire#w1
      Move(in := "IoScaling.S7Analog.Pt100.Climate.rScaledMin", out1 => #rScaledMin)
      Move(in := "IoScaling.S7Analog.Pt100.Climate.rScaledMax", out1 => #rScaledMax)
   END_RUNG
   // the same network as SCL:
   IF #iInSensorType = "IoScaling.S7Analog.Types.Pt100.Climate" THEN
       #iRawMin := "IoScaling.S7Analog.Pt100.Climate.iRawMin";
       #iRawMax := "IoScaling.S7Analog.Pt100.Climate.iRawMax";
       #rScaledMin := "IoScaling.S7Analog.Pt100.Climate.rScaledMin";
       #rScaledMax := "IoScaling.S7Analog.Pt100.Climate.rScaledMax";
   END_IF;
END_REGION

REGION Network 14: Ni100 RTD sensor type
   RUNG wire#powerrail
      { S7_Templates := "SrcType := Int" } EQ_Contact(in1 := #iInSensorType, in2 := "IoScaling.S7Analog.Types.Ni100")
      wire#w1
      Move(in := "IoScaling.S7Analog.Ni100.iRawMin", out1 => #iRawMin)
      Move(in := "IoScaling.S7Analog.Ni100.iRawMax", out1 => #iRawMax)
   END_RUNG
   RUNG wire#w1
      Move(in := "IoScaling.S7Analog.Ni100.rScaledMin", out1 => #rScaledMin)
      Move(in := "IoScaling.S7Analog.Ni100.rScaledMax", out1 => #rScaledMax)
   END_RUNG
   // the same network as SCL:
   IF #iInSensorType = "IoScaling.S7Analog.Types.Ni100" THEN
       #iRawMin := "IoScaling.S7Analog.Ni100.iRawMin";
       #iRawMax := "IoScaling.S7Analog.Ni100.iRawMax";
       #rScaledMin := "IoScaling.S7Analog.Ni100.rScaledMin";
       #rScaledMax := "IoScaling.S7Analog.Ni100.rScaledMax";
   END_IF;
END_REGION

REGION Network 15: Ni100 Climate RTD sensor type
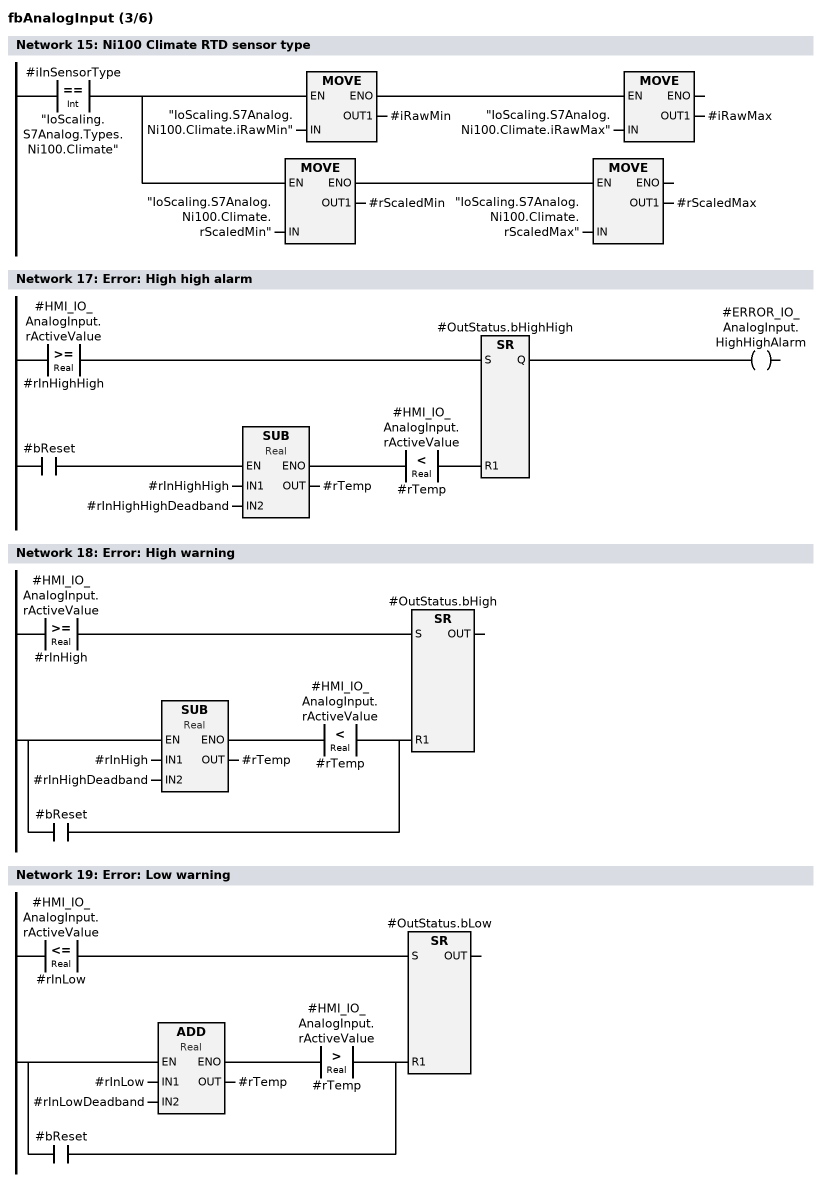
   RUNG wire#powerrail
      { S7_Templates := "SrcType := Int" } EQ_Contact(in1 := #iInSensorType, in2 := "IoScaling.S7Analog.Types.Ni100.Climate")
      wire#w1
      Move(in := "IoScaling.S7Analog.Ni100.Climate.iRawMin", out1 => #iRawMin)
      Move(in := "IoScaling.S7Analog.Ni100.Climate.iRawMax", out1 => #iRawMax)
   END_RUNG
   RUNG wire#w1
      Move(in := "IoScaling.S7Analog.Ni100.Climate.rScaledMin", out1 => #rScaledMin)
      Move(in := "IoScaling.S7Analog.Ni100.Climate.rScaledMax", out1 => #rScaledMax)
   END_RUNG
   // the same network as SCL:
   IF #iInSensorType = "IoScaling.S7Analog.Types.Ni100.Climate" THEN
       #iRawMin := "IoScaling.S7Analog.Ni100.Climate.iRawMin";
       #iRawMax := "IoScaling.S7Analog.Ni100.Climate.iRawMax";
       #rScaledMin := "IoScaling.S7Analog.Ni100.Climate.rScaledMin";
       #rScaledMax := "IoScaling.S7Analog.Ni100.Climate.rScaledMax";
   END_IF;
END_REGION

REGION Network 16: --------------------------------------------------------- Errors ------------------------------------------------------------------
END_REGION

REGION Network 17: Error: High high alarm
   RUNG wire#powerrail
      { S7_Templates := "SrcType := Real" } GE_Contact(in1 := #HMI_IO_AnalogInput.rActiveValue, in2 := #rInHighHigh)
      S_SR(operand := #OutStatus.bHighHigh, r1 := wire#w1)
      Coil( #ERROR_IO_AnalogInput.HighHighAlarm )
   END_RUNG
   RUNG wire#powerrail
      Contact( #bReset )
      { S7_Templates := "SrcType := Real" } Sub(in1 := #rInHighHigh, in2 := #rInHighHighDeadband, out => #rTemp)
      { S7_Templates := "SrcType := Real" } LT_Contact(in1 := #HMI_IO_AnalogInput.rActiveValue, in2 := #rTemp)
   END_RUNG wire#w1
   // the same network as SCL:
   IF #bReset THEN #rTemp := #rInHighHigh - #rInHighHighDeadband; END_IF;
   IF #HMI_IO_AnalogInput.rActiveValue >= #rInHighHigh THEN
       #OutStatus.bHighHigh := TRUE;   // SR flip-flop
   END_IF;
   IF #bReset AND (#HMI_IO_AnalogInput.rActiveValue < #rTemp) THEN #OutStatus.bHighHigh := FALSE; END_IF;
   #ERROR_IO_AnalogInput.HighHighAlarm := #OutStatus.bHighHigh;
END_REGION

REGION Network 18: Error: High warning
   RUNG wire#powerrail
      { S7_Templates := "SrcType := Real" } GE_Contact(in1 := #HMI_IO_AnalogInput.rActiveValue, in2 := #rInHigh)
      S_SR(operand := #OutStatus.bHigh, r1 := wire#w1)
   END_RUNG
   RUNG wire#powerrail
      { S7_Templates := "SrcType := Real" } Sub(in1 := #rInHigh, in2 := #rInHighDeadband, out => #rTemp)
      { S7_Templates := "SrcType := Real" } LT_Contact(in1 := #HMI_IO_AnalogInput.rActiveValue, in2 := #rTemp)
   END_RUNG wire#w1
   RUNG wire#powerrail
      Contact( #bReset )
   END_RUNG wire#w1
   // the same network as SCL:
   #rTemp := #rInHigh - #rInHighDeadband;
   IF #HMI_IO_AnalogInput.rActiveValue >= #rInHigh THEN
       #OutStatus.bHigh := TRUE;   // SR flip-flop
   END_IF;
   IF (#HMI_IO_AnalogInput.rActiveValue < #rTemp) OR #bReset THEN #OutStatus.bHigh := FALSE; END_IF;
END_REGION

REGION Network 19: Error: Low warning
   RUNG wire#powerrail
      { S7_Templates := "SrcType := Real" } LE_Contact(in1 := #HMI_IO_AnalogInput.rActiveValue, in2 := #rInLow)
      S_SR(operand := #OutStatus.bLow, r1 := wire#w1)
   END_RUNG
   RUNG wire#powerrail
      { S7_Templates := "SrcType := Real" } Add(in1 := #rInLow, in2 := #rInLowDeadband, out => #rTemp)
      { S7_Templates := "SrcType := Real" } GT_Contact(in1 := #HMI_IO_AnalogInput.rActiveValue, in2 := #rTemp)
   END_RUNG wire#w1
   RUNG wire#powerrail
      Contact( #bReset )
   END_RUNG wire#w1
   // the same network as SCL:
   #rTemp := #rInLow + #rInLowDeadband;
   IF #HMI_IO_AnalogInput.rActiveValue <= #rInLow THEN
       #OutStatus.bLow := TRUE;   // SR flip-flop
   END_IF;
   IF (#HMI_IO_AnalogInput.rActiveValue > #rTemp) OR #bReset THEN #OutStatus.bLow := FALSE; END_IF;
END_REGION

REGION Network 20: Error: Low low alarm
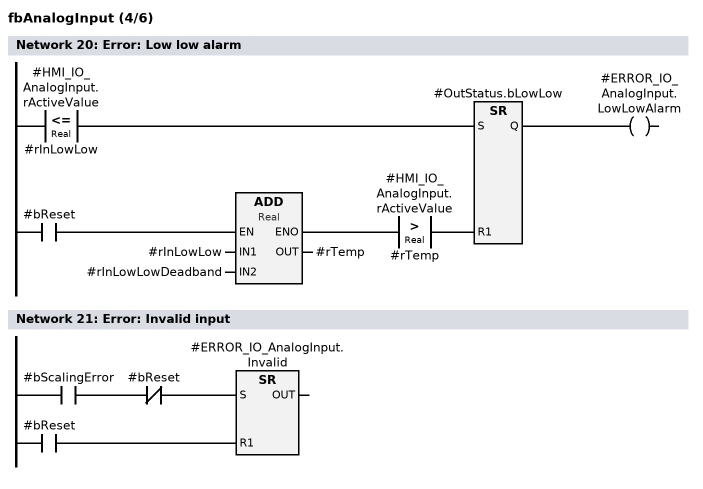
   RUNG wire#powerrail
      { S7_Templates := "SrcType := Real" } LE_Contact(in1 := #HMI_IO_AnalogInput.rActiveValue, in2 := #rInLowLow)
      S_SR(operand := #OutStatus.bLowLow, r1 := wire#w1)
      Coil( #ERROR_IO_AnalogInput.LowLowAlarm )
   END_RUNG
   RUNG wire#powerrail
      Contact( #bReset )
      { S7_Templates := "SrcType := Real" } Add(in1 := #rInLowLow, in2 := #rInLowLowDeadband, out => #rTemp)
      { S7_Templates := "SrcType := Real" } GT_Contact(in1 := #HMI_IO_AnalogInput.rActiveValue, in2 := #rTemp)
   END_RUNG wire#w1
   // the same network as SCL:
   IF #bReset THEN #rTemp := #rInLowLow + #rInLowLowDeadband; END_IF;
   IF #HMI_IO_AnalogInput.rActiveValue <= #rInLowLow THEN
       #OutStatus.bLowLow := TRUE;   // SR flip-flop
   END_IF;
   IF #bReset AND (#HMI_IO_AnalogInput.rActiveValue > #rTemp) THEN #OutStatus.bLowLow := FALSE; END_IF;
   #ERROR_IO_AnalogInput.LowLowAlarm := #OutStatus.bLowLow;
END_REGION

REGION Network 21: Error: Invalid input
   RUNG wire#powerrail
      Contact( #bScalingError )
      I_Contact( #bReset )
      S_SR(operand := #ERROR_IO_AnalogInput.Invalid, r1 := wire#w1)
   END_RUNG
   RUNG wire#powerrail
      Contact( #bReset )
   END_RUNG wire#w1
   // the same network as SCL:
   IF #bScalingError AND NOT #bReset THEN
       #ERROR_IO_AnalogInput.Invalid := TRUE;   // SR flip-flop
   END_IF;
   IF #bReset THEN #ERROR_IO_AnalogInput.Invalid := FALSE; END_IF;
END_REGION

REGION Network 22: Scroll errors on the HMI
   // Call the Error-Scroller which cyles through all possible errors and checks 
   // their state for display on the HMI
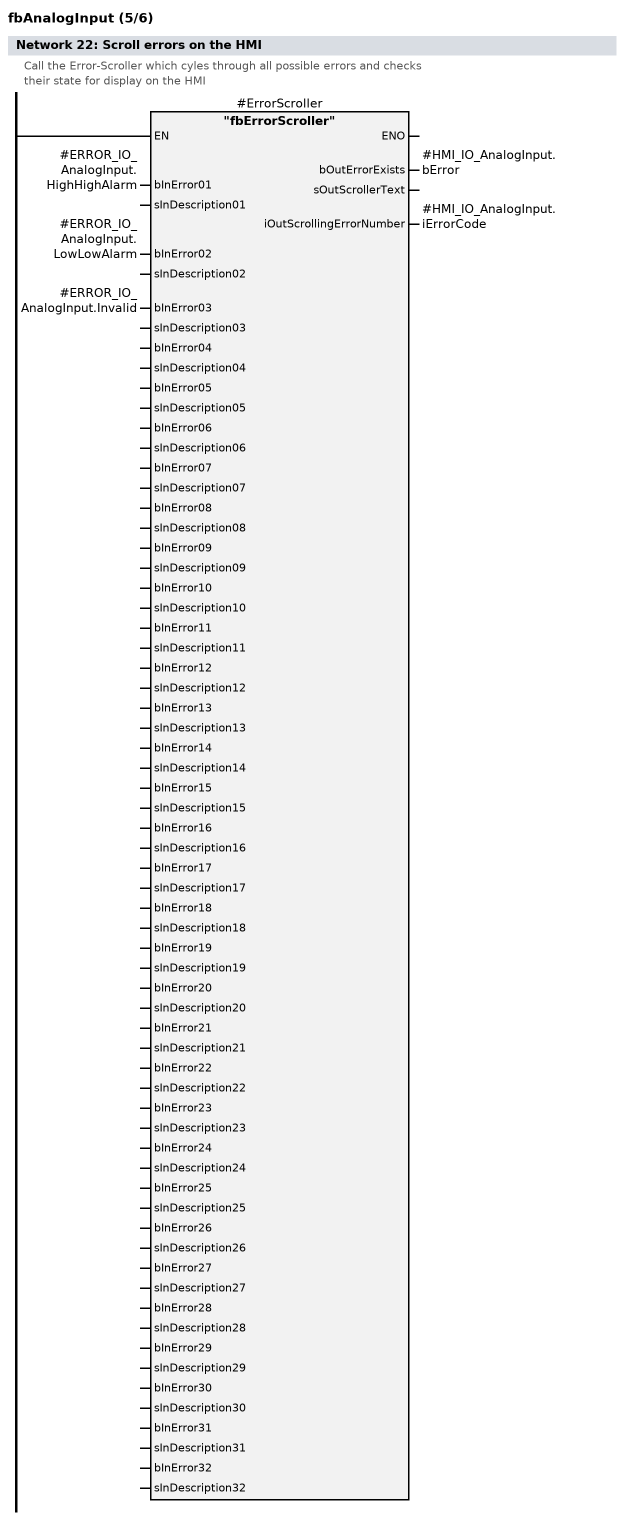
   RUNG wire#powerrail
      #ErrorScroller(bInError01 := #ERROR_IO_AnalogInput.HighHighAlarm, sInDescription01 :=, bInError02 := #ERROR_IO_AnalogInput.LowLowAlarm, sInDescription02 :=, bInError03 := #ERROR_IO_AnalogInput.Invalid, sInDescription03 :=, bInError04 :=, sInDescription04 :=, bInError05 :=, sInDescription05 :=, bInError06 :=, sInDescription06 :=, bInError07 :=, sInDescription07 :=, bInError08 :=, sInDescription08 :=, bInError09 :=, sInDescription09 :=, bInError10 :=, sInDescription10 :=, bInError11 :=, sInDescription11 :=, bInError12 :=, sInDescription12 :=, bInError13 :=, sInDescription13 :=, bInError14 :=, sInDescription14 :=, bInError15 :=, sInDescription15 :=, bInError16 :=, sInDescription16 :=, bInError17 :=, sInDescription17 :=, bInError18 :=, sInDescription18 :=, bInError19 :=, sInDescription19 :=, bInError20 :=, sInDescription20 :=, bInError21 :=, sInDescription21 :=, bInError22 :=, sInDescription22 :=, bInError23 :=, sInDescription23 :=, bInError24 :=, sInDescription24 :=, bInError25 :=, sInDescription25 :=, bInError26 :=, sInDescription26 :=, bInError27 :=, sInDescription27 :=, bInError28 :=, sInDescription28 :=, bInError29 :=, sInDescription29 :=, bInError30 :=, sInDescription30 :=, bInError31 :=, sInDescription31 :=, bInError32 :=, sInDescription32 :=, bOutErrorExists => #HMI_IO_AnalogInput.bError, sOutScrollerText =>, iOutScrollingErrorNumber => #HMI_IO_AnalogInput.iErrorCode)
   END_RUNG
   // the same network as SCL:
   #ErrorScroller(bInError01 := #ERROR_IO_AnalogInput.HighHighAlarm,   // "fbErrorScroller"
                  bInError02 := #ERROR_IO_AnalogInput.LowLowAlarm,
                  bInError03 := #ERROR_IO_AnalogInput.Invalid,
                  bOutErrorExists => #HMI_IO_AnalogInput.bError,
                  iOutScrollingErrorNumber => #HMI_IO_AnalogInput.iErrorCode);
END_REGION

REGION Network 23: Set HMI Status
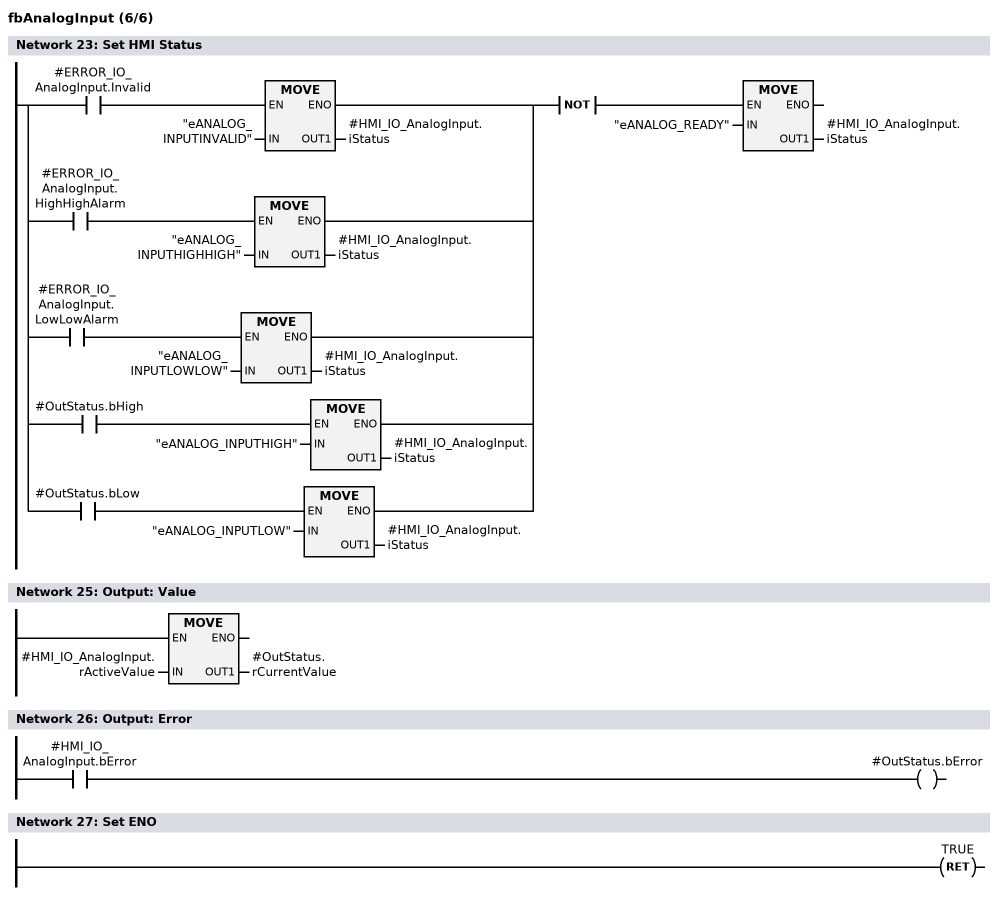
   RUNG wire#powerrail
      Contact( #ERROR_IO_AnalogInput.Invalid )
      Move(in := "eANALOG_INPUTINVALID", out1 => #HMI_IO_AnalogInput.iStatus)
      wire#w1
      Not()
      Move(in := "eANALOG_READY", out1 => #HMI_IO_AnalogInput.iStatus)
   END_RUNG
   RUNG wire#powerrail
      Contact( #ERROR_IO_AnalogInput.HighHighAlarm )
      Move(in := "eANALOG_INPUTHIGHHIGH", out1 => #HMI_IO_AnalogInput.iStatus)
   END_RUNG wire#w1
   RUNG wire#powerrail
      Contact( #ERROR_IO_AnalogInput.LowLowAlarm )
      Move(in := "eANALOG_INPUTLOWLOW", out1 => #HMI_IO_AnalogInput.iStatus)
   END_RUNG wire#w1
   RUNG wire#powerrail
      Contact( #OutStatus.bHigh )
      Move(in := "eANALOG_INPUTHIGH", out1 => #HMI_IO_AnalogInput.iStatus)
   END_RUNG wire#w1
   RUNG wire#powerrail
      Contact( #OutStatus.bLow )
      Move(in := "eANALOG_INPUTLOW", out1 => #HMI_IO_AnalogInput.iStatus)
   END_RUNG wire#w1
   // the same network as SCL:
   IF #ERROR_IO_AnalogInput.Invalid THEN #HMI_IO_AnalogInput.iStatus := "eANALOG_INPUTINVALID"; END_IF;
   IF #ERROR_IO_AnalogInput.HighHighAlarm THEN
       #HMI_IO_AnalogInput.iStatus := "eANALOG_INPUTHIGHHIGH";
   END_IF;
   IF #ERROR_IO_AnalogInput.LowLowAlarm THEN #HMI_IO_AnalogInput.iStatus := "eANALOG_INPUTLOWLOW"; END_IF;
   IF #OutStatus.bHigh THEN #HMI_IO_AnalogInput.iStatus := "eANALOG_INPUTHIGH"; END_IF;
   IF #OutStatus.bLow THEN #HMI_IO_AnalogInput.iStatus := "eANALOG_INPUTLOW"; END_IF;
   IF NOT (#ERROR_IO_AnalogInput.Invalid OR #ERROR_IO_AnalogInput.HighHighAlarm OR #ERROR_IO_AnalogInput.LowLowAlarm OR #OutStatus.bHigh OR #OutStatus.bLow) THEN
       #HMI_IO_AnalogInput.iStatus := "eANALOG_READY";
   END_IF;
END_REGION

REGION Network 24: --------------------------------------------------------- Outputs ------------------------------------------------------------------
END_REGION

REGION Network 25: Output: Value
   RUNG wire#powerrail
      Move(in := #HMI_IO_AnalogInput.rActiveValue, out1 => #OutStatus.rCurrentValue)
   END_RUNG
   // the same network as SCL:
   #OutStatus.rCurrentValue := #HMI_IO_AnalogInput.rActiveValue;
END_REGION

REGION Network 26: Output: Error
   RUNG wire#powerrail
      Contact( #HMI_IO_AnalogInput.bError )
      Coil( #OutStatus.bError )
   END_RUNG
   // the same network as SCL:
   #OutStatus.bError := #HMI_IO_AnalogInput.bError;
END_REGION

REGION Network 27: Set ENO
   RUNG wire#powerrail
      ReturnCoil( TRUE )
   END_RUNG
   // the same network as SCL:
   ENO := TRUE;
   RETURN;
END_REGION
END_FUNCTION_BLOCK

FUNCTION_BLOCK "fbDigitalOutput"   // FB146, LAD
TITLE = Controls a digital output
{ S7_Optimized_Access := 'TRUE' }
VERSION : 0.1
   VAR_INPUT
      iInMode : Int;   // Current mode
      bInEstop : Bool;   // System e-stop exists
      bInEnable : Bool;   // Enables the digital output
      bInCommand : Bool;   // Auto mode value of output
   END_VAR
   VAR_OUTPUT
      bOutCommand : Bool;   // Actual analog output value
   END_VAR
   VAR_IN_OUT
      HMI_IO_DigitalOutput : "udtHMI_DigitalOutput";   // HMI control strucure for a digital output
   END_VAR
   VAR
      bCommand : Bool;
      PB : Struct
         bOn : Bool;
         bOff : Bool;
      END_STRUCT;
   END_VAR
   VAR_TEMP   // added for the SCL form of the ladder/FBD networks
      _w1 : Bool;
      _w2 : Bool;
   END_VAR
BEGIN

REGION Network 1: --------------------------------------------------------- Inputs ------------------------------------------------------------------
END_REGION

REGION Network 2: Read in auto mode value
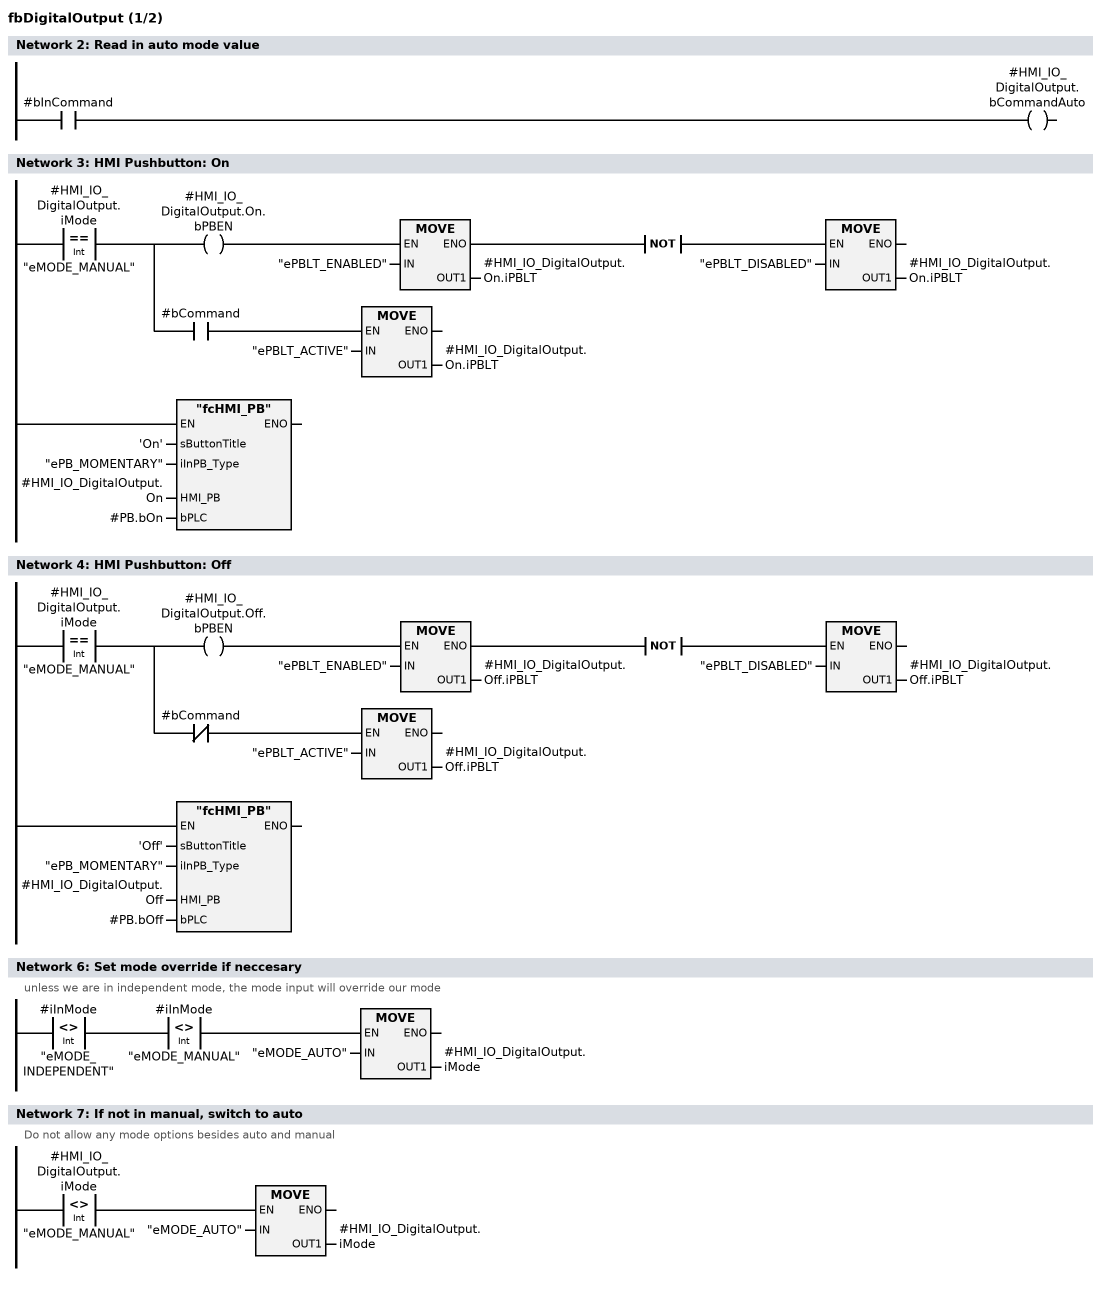
   RUNG wire#powerrail
      Contact( #bInCommand )
      Coil( #HMI_IO_DigitalOutput.bCommandAuto )
   END_RUNG
   // the same network as SCL:
   #HMI_IO_DigitalOutput.bCommandAuto := #bInCommand;
END_REGION

REGION Network 3: HMI Pushbutton: On
   RUNG wire#powerrail
      { S7_Templates := "SrcType := Int" } EQ_Contact(in1 := #HMI_IO_DigitalOutput.iMode, in2 := "eMODE_MANUAL")
      wire#w1
      Coil( #HMI_IO_DigitalOutput.On.bPBEN )
      Move(in := "ePBLT_ENABLED", out1 => #HMI_IO_DigitalOutput.On.iPBLT)
      Not()
      Move(in := "ePBLT_DISABLED", out1 => #HMI_IO_DigitalOutput.On.iPBLT)
   END_RUNG
   RUNG wire#w1
      Contact( #bCommand )
      Move(in := "ePBLT_ACTIVE", out1 => #HMI_IO_DigitalOutput.On.iPBLT)
   END_RUNG
   RUNG wire#powerrail
      "fcHMI_PB"(sButtonTitle := 'On', iInPB_Type := "ePB_MOMENTARY", HMI_PB := #HMI_IO_DigitalOutput.On, bPLC := #PB.bOn)
   END_RUNG
   // the same network as SCL:
   #HMI_IO_DigitalOutput.On.bPBEN := #HMI_IO_DigitalOutput.iMode = "eMODE_MANUAL";
   IF #HMI_IO_DigitalOutput.On.bPBEN THEN #HMI_IO_DigitalOutput.On.iPBLT := "ePBLT_ENABLED"; END_IF;
   IF NOT #HMI_IO_DigitalOutput.On.bPBEN THEN #HMI_IO_DigitalOutput.On.iPBLT := "ePBLT_DISABLED"; END_IF;
   IF #HMI_IO_DigitalOutput.On.bPBEN AND #bCommand THEN
       #HMI_IO_DigitalOutput.On.iPBLT := "ePBLT_ACTIVE";
   END_IF;
   "fcHMI_PB"(sButtonTitle := 'On',
              iInPB_Type := "ePB_MOMENTARY",
              HMI_PB := #HMI_IO_DigitalOutput.On,
              bPLC := #PB.bOn);
END_REGION

REGION Network 4: HMI Pushbutton: Off
   RUNG wire#powerrail
      { S7_Templates := "SrcType := Int" } EQ_Contact(in1 := #HMI_IO_DigitalOutput.iMode, in2 := "eMODE_MANUAL")
      wire#w1
      Coil( #HMI_IO_DigitalOutput.Off.bPBEN )
      Move(in := "ePBLT_ENABLED", out1 => #HMI_IO_DigitalOutput.Off.iPBLT)
      Not()
      Move(in := "ePBLT_DISABLED", out1 => #HMI_IO_DigitalOutput.Off.iPBLT)
   END_RUNG
   RUNG wire#w1
      I_Contact( #bCommand )
      Move(in := "ePBLT_ACTIVE", out1 => #HMI_IO_DigitalOutput.Off.iPBLT)
   END_RUNG
   RUNG wire#powerrail
      "fcHMI_PB"(sButtonTitle := 'Off', iInPB_Type := "ePB_MOMENTARY", HMI_PB := #HMI_IO_DigitalOutput.Off, bPLC := #PB.bOff)
   END_RUNG
   // the same network as SCL:
   #HMI_IO_DigitalOutput.Off.bPBEN := #HMI_IO_DigitalOutput.iMode = "eMODE_MANUAL";
   IF #HMI_IO_DigitalOutput.Off.bPBEN THEN #HMI_IO_DigitalOutput.Off.iPBLT := "ePBLT_ENABLED"; END_IF;
   IF NOT #HMI_IO_DigitalOutput.Off.bPBEN THEN #HMI_IO_DigitalOutput.Off.iPBLT := "ePBLT_DISABLED"; END_IF;
   IF #HMI_IO_DigitalOutput.Off.bPBEN AND NOT #bCommand THEN
       #HMI_IO_DigitalOutput.Off.iPBLT := "ePBLT_ACTIVE";
   END_IF;
   "fcHMI_PB"(sButtonTitle := 'Off',
              iInPB_Type := "ePB_MOMENTARY",
              HMI_PB := #HMI_IO_DigitalOutput.Off,
              bPLC := #PB.bOff);
END_REGION

REGION Network 5: --------------------------------------------------- Control Logic ------------------------------------------------------------
END_REGION

REGION Network 6: Set mode override if neccesary
   // unless we are in independent mode, the mode input will override our mode
   RUNG wire#powerrail
      { S7_Templates := "SrcType := Int" } NE_Contact(in1 := #iInMode, in2 := "eMODE_INDEPENDENT")
      { S7_Templates := "SrcType := Int" } NE_Contact(in1 := #iInMode, in2 := "eMODE_MANUAL")
      Move(in := "eMODE_AUTO", out1 => #HMI_IO_DigitalOutput.iMode)
   END_RUNG
   // the same network as SCL:
   IF (#iInMode <> "eMODE_INDEPENDENT") AND (#iInMode <> "eMODE_MANUAL") THEN
       #HMI_IO_DigitalOutput.iMode := "eMODE_AUTO";
   END_IF;
END_REGION

REGION Network 7: If not in manual, switch to auto
   // Do not allow any mode options besides auto and manual
   RUNG wire#powerrail
      { S7_Templates := "SrcType := Int" } NE_Contact(in1 := #HMI_IO_DigitalOutput.iMode, in2 := "eMODE_MANUAL")
      Move(in := "eMODE_AUTO", out1 => #HMI_IO_DigitalOutput.iMode)
   END_RUNG
   // the same network as SCL:
   IF #HMI_IO_DigitalOutput.iMode <> "eMODE_MANUAL" THEN #HMI_IO_DigitalOutput.iMode := "eMODE_AUTO"; END_IF;
END_REGION

REGION Network 8: Determine if manual or auto mode is active
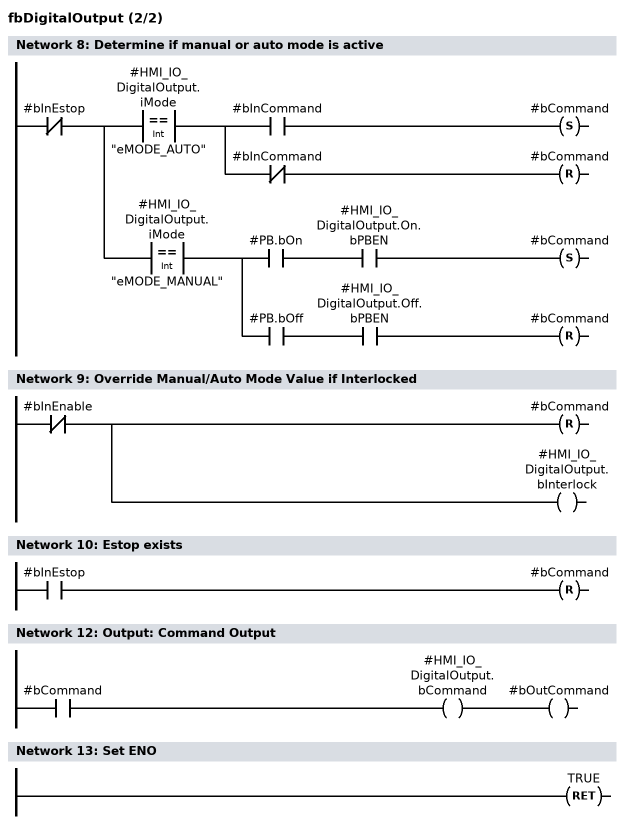
   RUNG wire#powerrail
      I_Contact( #bInEstop )
      wire#w1
      { S7_Templates := "SrcType := Int" } EQ_Contact(in1 := #HMI_IO_DigitalOutput.iMode, in2 := "eMODE_AUTO")
      wire#w2
      Contact( #bInCommand )
      S_Coil( #bCommand )
   END_RUNG
   RUNG wire#w2
      I_Contact( #bInCommand )
      R_Coil( #bCommand )
   END_RUNG
   RUNG wire#w1
      { S7_Templates := "SrcType := Int" } EQ_Contact(in1 := #HMI_IO_DigitalOutput.iMode, in2 := "eMODE_MANUAL")
      wire#w3
      Contact( #PB.bOn )
      Contact( #HMI_IO_DigitalOutput.On.bPBEN )
      S_Coil( #bCommand )
   END_RUNG
   RUNG wire#w3
      Contact( #PB.bOff )
      Contact( #HMI_IO_DigitalOutput.Off.bPBEN )
      R_Coil( #bCommand )
   END_RUNG
   // the same network as SCL:
   #_w1 := NOT #bInEstop AND (#HMI_IO_DigitalOutput.iMode = "eMODE_AUTO");
   IF #_w1 AND #bInCommand THEN #bCommand := TRUE; END_IF;
   IF #_w1 AND NOT #bInCommand THEN #bCommand := FALSE; END_IF;
   #_w2 := NOT #bInEstop AND (#HMI_IO_DigitalOutput.iMode = "eMODE_MANUAL");
   IF #_w2 AND #PB.bOn AND #HMI_IO_DigitalOutput.On.bPBEN THEN #bCommand := TRUE; END_IF;
   IF #_w2 AND #PB.bOff AND #HMI_IO_DigitalOutput.Off.bPBEN THEN #bCommand := FALSE; END_IF;
END_REGION

REGION Network 9: Override Manual/Auto Mode Value if Interlocked
   RUNG wire#powerrail
      I_Contact( #bInEnable )
      wire#w1
      R_Coil( #bCommand )
   END_RUNG
   RUNG wire#w1
      Coil( #HMI_IO_DigitalOutput.bInterlock )
   END_RUNG
   // the same network as SCL:
   IF NOT #bInEnable THEN #bCommand := FALSE; END_IF;
   #HMI_IO_DigitalOutput.bInterlock := NOT #bInEnable;
END_REGION

REGION Network 10: Estop exists
   RUNG wire#powerrail
      Contact( #bInEstop )
      R_Coil( #bCommand )
   END_RUNG
   // the same network as SCL:
   IF #bInEstop THEN #bCommand := FALSE; END_IF;
END_REGION

REGION Network 11: --------------------------------------------------------- Outputs ------------------------------------------------------------------
END_REGION

REGION Network 12: Output: Command Output
   RUNG wire#powerrail
      Contact( #bCommand )
      Coil( #HMI_IO_DigitalOutput.bCommand )
      Coil( #bOutCommand )
   END_RUNG
   // the same network as SCL:
   #HMI_IO_DigitalOutput.bCommand := #bCommand;
   #bOutCommand := #bCommand;
END_REGION

REGION Network 13: Set ENO
   RUNG wire#powerrail
      ReturnCoil( TRUE )
   END_RUNG
   // the same network as SCL:
   ENO := TRUE;
   RETURN;
END_REGION
END_FUNCTION_BLOCK

FUNCTION_BLOCK "fbDigitalInput"   // FB211, LAD
TITLE = Debounces a digital sensor
{ S7_Optimized_Access := 'TRUE' }
AUTHOR : JRM
VERSION : 0.1
   VAR_INPUT
      iInMode : Int;   // Current mode
      bInInput : Bool;   // Actual digital input tag
      tInOnDebounce : Time;   // Debounce time for input TRUE
      tInOffDebounce : Time;   // Debounce time for input FALSE
   END_VAR
   VAR_OUTPUT
      OutStatus : "udtStatus_DigitalInput";   // Digital Input Status
   END_VAR
   VAR_IN_OUT
      HMI_IO_DigitalInput : "udtHMI_DigitalInput";   // HMI control structure for digital input
   END_VAR
   VAR
      TON_On : IEC_TIMER;   // Timer for ON debounce
      TON_Off : IEC_TIMER;   // Timer for OFF debounce
      PB : Struct   // HMI Simulation Pushbuttons
         bOn : Bool;   // Simulate On
         bOff : Bool;   // Simulate Off
      END_STRUCT;
      bTON_On : Bool;   // ON debounce timer complete
      bTON_Off : Bool;   // OFF debounce timer complete
      FP_On : Bool;   // Rising edge memory bit
      FN_Off : Bool;   // Falling edge memory bit
   END_VAR
   VAR_TEMP   // added for the SCL form of the ladder/FBD networks
      _w1 : Bool;
      _w2 : Bool;
   END_VAR
BEGIN

REGION Network 1: --------------------------------------------------------- Inputs ------------------------------------------------------------------
END_REGION

REGION Network 2: HMI Pushbutton: On
